	// Search correlating zone
	// Check from target window to the left until MaxFrontedgeDeviation
	ELSE
		// Calculate max number of allowed front deviation windows
		NumberOfDeviationWindows := UDINT_TO_UINT(mMaxFrontEdgeDeviation / WindowSize);
		
		// Add an additional window if rest of division was unequal 0
		IF mMaxFrontEdgeDeviation MOD WindowSize > 0 THEN
			NumberOfDeviationWindows := NumberOfDeviationWindows + 1;
		END_IF
		
		// Get max tracking position for valid zone
		MaxTrackingPosition := M_GetTrackingPosition(mAbsolutePosition - mMaxFrontEdgeDeviation);

		// Search for adjacent zone
		mWindowIndex := mNewWindowIndexFE;
				
		// Check all additional windows plus begin
		FOR mIdx := 1 TO NumberOfDeviationWindows + 1 DO
			// Correct window border overflow
			IF mWindowIndex > MaxWindowIndex THEN
				mWindowIndex := mWindowIndex - MaxWindowIndex;
			END_IF
			
			// Search next zone
			IF WindowTable[mWindowIndex].ZoneIndex > 0 THEN
				DistanceToTU_End := M_GetDistanceToTU_End(mAbsolutePosition, WindowTable[mWindowIndex].ZoneIndex);
				DistanceToTU_Start := M_GetDistanceToTU_Start(mAbsolutePosition, WindowTable[mWindowIndex].ZoneIndex);
			
				// When a found zone is valid, check if edge is in valid range
				IF WindowTable[mWindowIndex].State = E_WindowTrackingWindowState.Front_EDGE THEN
					// Check if it's not last deviation window to check
					IF mIdx < NumberOfDeviationWindows + 1 THEN
						// Return found zone
						ZoneIndex := WindowTable[mWindowIndex].ZoneIndex;
					ELSE
						// Check position in window for max deviation
						IF WindowTable[mWindowIndex].TU_FrontEdgePosition <= MaxTrackingPosition THEN			
							// Return found zone
							ZoneIndex := WindowTable[mWindowIndex].ZoneIndex;
						END_IF
					END_IF
					EXIT;
					
				// Ensure TU end has not passed resync position and TU begin has reacher in minimum MaxDeviation pos
				// Remark: >0 = It is infront of resync position 
				ELSIF DistanceToTU_End > 0 AND
					  DistanceToTU_Start <= UDINT_TO_DINT(mMaxFrontEdgeDeviation) THEN
					// Return found zone
					ZoneIndex := WindowTable[mWindowIndex].ZoneIndex;
					EXIT;
				END_IF
			END_IF
			
			mWindowIndex := mWindowIndex + 1;
		END_FOR 
	END_IF
END_IF

// Ensure zone is valid (Consists of a TU, adaption of FE possible)
IF ZoneIndex > 0 THEN
	// Only possible if zone consists of a physical TU
	IF ZoneTable[ZoneIndex].TU_Present THEN
		// Ensure that no other zone is between new front edge and old rear edge
		mWindowIndex := mNewWindowIndexFE;
		ResyncPossible := TRUE;
		
		// Calculate new zone length in windows
		IF ZoneTable[ZoneIndex].ZoneEndWindowIndex > mNewWindowIndexFE THEN
			mNewZoneWindowLength := ZoneTable[ZoneIndex].ZoneEndWindowIndex - mNewWindowIndexFE + 1;
		ELSE
			mNewZoneWindowLength := ZoneTable[ZoneIndex].ZoneEndWindowIndex + MaxWindowIndex - mNewWindowIndexFE + 1;
		END_IF
	
		// Ensure resync has space
		FOR mIdx := 1 TO mNewZoneWindowLength DO	
			// If found window is empty or already part of the zone
			IF WindowTable[mWindowIndex].ZoneIndex = 0 OR
			   WindowTable[mWindowIndex].ZoneIndex = ZoneIndex THEN
			   // Window is valid
			   ;
			
			// Otherwise another zone is found, try to shift
			ELSE
				mZoneFreeOk := M_MakeSpace(
									mStartWindowIndex 	:= mWindowIndex, 
									mWindowsToFree 		:= 1,
									mAllowZoneDelete 	:= TRUE);
									
				IF NOT mZoneFreeOk THEN
					// Error, zone could not be shifted -> abort
					ResyncPossible := FALSE;
					EXIT;
				END_IF
			END_IF
			  
			mWindowIndex := mWindowIndex + 1;

			// Correct window border overflow
			IF mWindowIndex > MaxWindowIndex THEN
				mWindowIndex := mWindowIndex - MaxWindowIndex;
			END_IF
		END_FOR  
	END_IF
END_IF

// Process when a valid zone could be found
IF ZoneIndex > 0 AND ResyncPossible THEN
	// Calculate length of existing zone in windows
	IF ZoneTable[ZoneIndex].ZoneEndWindowIndex > ZoneTable[ZoneIndex].ZoneStartWindowIndex THEN
		ZoneWindowLength := ZoneTable[ZoneIndex].ZoneEndWindowIndex - ZoneTable[ZoneIndex].ZoneStartWindowIndex + 1;
	ELSE
		ZoneWindowLength := ZoneTable[ZoneIndex].ZoneEndWindowIndex + MaxWindowIndex  - ZoneTable[ZoneIndex].ZoneStartWindowIndex + 1;
	END_IF
	
	// Get existing front edge window
	ExistingWindowIndexFE := ZoneTable[ZoneIndex].TU_StartWindowIndex;
		
	// When front edge window could be found
	IF ExistingWindowIndexFE > 0 THEN
		// Store old window, because its possible to overwrite existing position
		OldWindowFE := WindowTable[ExistingWindowIndexFE];
		M_ClearWindow(ExistingWindowIndexFE);
		
		// Copy old window to new
		WindowTable[mNewWindowIndexFE] := OldWindowFE;
		
		NewPositionFE := M_GetTrackingPosition(mAbsolutePosition);
		
		// Adapt edge position and zone length
		WindowTable[mNewWindowIndexFE].TU_FrontEdgePosition := NewPositionFE;
		ZoneTable[ZoneIndex].ZoneStartWindowIndex := mNewWindowIndexFE;
		ZoneTable[ZoneIndex].TU_StartWindowIndex := mNewWindowIndexFE;
		ZoneTable[ZoneIndex].ZoneStartPosition := NewPositionFE;
		
		IF ZoneTable[ZoneIndex].ZoneEndPosition >= ZoneTable[ZoneIndex].ZoneStartPosition THEN
			ZoneTable[ZoneIndex].ZoneLength := UDINT_TO_UINT(ZoneTable[ZoneIndex].ZoneEndPosition - ZoneTable[ZoneIndex].ZoneStartPosition);
		ELSE
			ZoneTable[ZoneIndex].ZoneLength := UDINT_TO_UINT(ZoneTable[ZoneIndex].ZoneEndPosition + TotalTrackingLength - ZoneTable[ZoneIndex].ZoneStartPosition);
		END_IF

		// Clean all windows to the right of this zone
		mWindowIndex := mNewWindowIndexFE - 1;
		
		FOR mIdx := 1 TO MaxWindowIndex DO	
			// Correct window border overflow
			IF mWindowIndex <= 0 THEN
				mWindowIndex := mWindowIndex + MaxWindowIndex;
			END_IF
			
			// When window right of the front edge is part of the same zone, clean it
			IF WindowTable[mWindowIndex].ZoneIndex = ZoneIndex THEN
				M_ClearWindow(mWindowIndex);
				mWindowIndex := mWindowIndex -1;
			// Otherwise no other windows to clean
			ELSE
				EXIT;
			END_IF
		END_FOR  
			
		// Fill gap windows to the left
		mWindowIndex := mNewWindowIndexFE;
				
		FOR mIdx := 1 TO mNewZoneWindowLength DO	
			// Correct window border overflow
			IF mWindowIndex > MaxWindowIndex THEN
				mWindowIndex := mWindowIndex - MaxWindowIndex;
			END_IF
			
			// Assign ZoneIndex to all windows
			WindowTable[mWindowIndex].ZoneIndex := ZoneIndex;
			
			// Overwrite all windows as occupied except begin and end
			IF WindowTable[mWindowIndex].State = E_WindowTrackingWindowState.FRONT_EDGE THEN
				;
			// Stop overwriting at rear edge window
            ELSIF WindowTable[mWindowIndex].State = E_WindowTrackingWindowState.REAR_EDGE THEN
				EXIT;
			ELSE
				// Assign ZoneIndex to all windows
				WindowTable[mWindowIndex].ZoneIndex := ZoneIndex;
				WindowTable[mWindowIndex].State := E_WindowTrackingWindowState.OCCUPIED;
			
				// Possible flush can be resettet, because of synchronization its valid again
				WindowTable[mWindowIndex].Flush := 0;
				WindowTable[mWindowIndex].TU_FrontEdgePosition := 0;
				WindowTable[mWindowIndex].TU_RearEdgePosition := 0;
			END_IF

			mWindowIndex := mWindowIndex + 1;
		END_FOR  
		
		M_ResyncOnlyFE := ZoneIndex;
	END_IF
END_IF
END_METHOD

/// This function synchronize only Rear edge to a specific position and calculates new TU length.
/// Remark: Zone end gets adjusted to new rear edge position. Spare windows after rear edge get removed.
/// Remark: If at absolute position no zone is found, it search to the right
/// until "mMaxFrontEdgeDeviation" to find one to synchronize.
METHOD M_ResyncOnlyRE : UINT // Returns > 0 of the synchronized Zone index, otherwise 0
VAR_INPUT
	mAbsolutePosition		: UDINT; // Absolute position [mm]
	mMaxRearEdgeDeviation 	: UDINT; (* When zone can not be found at "Absolute position",
										a search upwards is executed to a limit of MaxRearEdgeDeviation [mm]*)
END_VAR
VAR_INST
	MinTrackingPosition		: UDINT; // Min tracking distance to search for a zone
	NumberOfDeviationWindows: UINT; // Number of windows for maximal edge deviation 
	ZoneIndex				: UINT; // Zone index
	ResyncPossible			: BOOL; // Resync is possible
	ExistingWindowIndexRE	: UINT; // Existing rear edge window index
	ZoneWindowLength 		: UINT; // Length of zone to be moved
	OldWindowRE				: ST_WindowTrackingWindow; // Stored old rear edge window
	NewPositionRE			: UDINT; // New rear edge position in tracking
	DistanceToTU_End		: DINT; // Distance to found TU End
	DistanceToTU_Start		: DINT; // Distance to found TU start
END_VAR
VAR
	mZoneFreeOk				: BOOL; // Successfully
	mNewZoneWindowLength	: UINT; // Length of windows of aligned zone
	mNewWindowIndexRE		: UINT; // Actual window index
	mWindowIndex			: UINT; // Window index iterator
	mIdx					: UINT; // Loop iterator
END_VAR
M_ResyncOnlyRE := 0;
ZoneIndex := 0;
NumberOfDeviationWindows := 0;

// Validate values
IF WindowSize = 0 THEN
	RETURN;
END_IF

// Get window index at position
mNewWindowIndexRE := M_GetWindowIndex(mAbsolutePosition);

IF mNewWindowIndexRE > 0 AND mNewWindowIndexRE <= WindowTracking.MAX_NUMBER_OF_WINDOWS THEN
	// Ensure that target window is not already a front edge window 
	// This is not permitted, minimum zone is two window
	IF WindowTable[mNewWindowIndexRE].State = E_WindowTrackingWindowState.FRONT_EDGE THEN
		ZoneIndex := 0;
		
	// Search correlating zone
	// Check from target window to the right until MaxFrontedgeDeviation
	ELSE
		// Calculate max number of allowed rear edge deviation windows
		NumberOfDeviationWindows := UDINT_TO_UINT(mMaxRearEdgeDeviation / WindowSize);
		
		// Add an additional window if rest of division was unequal 0
		IF mMaxRearEdgeDeviation MOD WindowSize > 0 THEN
			NumberOfDeviationWindows := NumberOfDeviationWindows + 1;
		END_IF
		
		// Get min  tracking position for valid zone
		MinTrackingPosition := M_GetTrackingPosition(mAbsolutePosition + mMaxRearEdgeDeviation);

		// Search for a adjacent zone
		mWindowIndex := mNewWindowIndexRE;

		FOR mIdx := 1 TO NumberOfDeviationWindows + 1 DO	
			// Correct window border overflow
			IF mWindowIndex <= 0 THEN
				mWindowIndex := mWindowIndex + MaxWindowIndex;
			END_IF
			
			// Search next zone
			IF WindowTable[mWindowIndex].ZoneIndex > 0 THEN
				DistanceToTU_End := M_GetDistanceToTU_End(mAbsolutePosition, WindowTable[mWindowIndex].ZoneIndex);
				DistanceToTU_Start := M_GetDistanceToTU_Start(mAbsolutePosition, WindowTable[mWindowIndex].ZoneIndex);
			
				// When a rear edge was found check for valid range
				IF WindowTable[mWindowIndex].State = E_WindowTrackingWindowState.REAR_EDGE THEN
					// If it's not last deviation window to check
					IF mIdx < NumberOfDeviationWindows + 1 THEN
						// Return found zone
						ZoneIndex := WindowTable[mWindowIndex].ZoneIndex;
					ELSE
						// Check position in window for max deviation
						IF WindowTable[mWindowIndex].TU_RearEdgePosition >= MinTrackingPosition THEN			
							// Return found zone
							ZoneIndex := WindowTable[mWindowIndex].ZoneIndex;
						END_IF
					END_IF
					EXIT;
					
				// Ensure TU start has passed resync position and TU end has reached in minimum MaxDeviation pos
				// Remark: >0 = It is infront of resync position 
				ELSIF DistanceToTU_Start < 0 AND
                      DistanceToTU_End >= UDINT_TO_DINT(mMaxRearEdgeDeviation) THEN
				   	// Return found zone
					ZoneIndex := WindowTable[mWindowIndex].ZoneIndex;
					EXIT;
				END_IF
			END_IF
			
			mWindowIndex := mWindowIndex - 1;
		END_FOR 
	END_IF
END_IF

// Ensure zone is valid (Consists of a TU, adaption of RE possible)
IF ZoneIndex > 0 THEN
	// Only possible if zone consists of a physical TU
	IF ZoneTable[ZoneIndex].TU_Present THEN
		// Ensure that no other zone is between new rear edge and old front edge
		mWindowIndex := ZoneTable[ZoneIndex].ZoneStartWindowIndex;
		ResyncPossible := TRUE;
		
		// Calculate new zone length in windows
		IF mNewWindowIndexRE > ZoneTable[ZoneIndex].ZoneStartWindowIndex THEN
			mNewZoneWindowLength := mNewWindowIndexRE - ZoneTable[ZoneIndex].ZoneStartWindowIndex + 1;
		ELSE
			mNewZoneWindowLength := mNewWindowIndexRE  + MaxWindowIndex - ZoneTable[ZoneIndex].ZoneStartWindowIndex + 1;
		END_IF
	
		// Validate that sync is possible
		FOR mIdx := 1 TO mNewZoneWindowLength DO	
			// If found window is empty or already part of the zone
			IF WindowTable[mWindowIndex].ZoneIndex = 0 OR
			   WindowTable[mWindowIndex].ZoneIndex = ZoneIndex THEN
			   // Window is valid
			   ;
			
			// Otherwise another zone is found, try to shift
			ELSE
				mZoneFreeOk := M_MakeSpace(
									mStartWindowIndex 	:= mWindowIndex, 
									mWindowsToFree 		:= 1,
									mAllowZoneDelete 	:= TRUE);
									
				IF NOT mZoneFreeOk THEN
					// Error, zone could not be shifted -> abort
					ResyncPossible := FALSE;
					EXIT;
				END_IF
			END_IF
			  
			mWindowIndex := mWindowIndex + 1;

			// Correct window border overflow
			IF mWindowIndex > MaxWindowIndex THEN
				mWindowIndex := mWindowIndex - MaxWindowIndex;
			END_IF
		END_FOR  
	END_IF
END_IF

IF ZoneIndex > 0 AND ResyncPossible THEN
	// Calculate length of existing zone in windows
	IF ZoneTable[ZoneIndex].ZoneEndWindowIndex > ZoneTable[ZoneIndex].ZoneStartWindowIndex THEN
		ZoneWindowLength := ZoneTable[ZoneIndex].ZoneEndWindowIndex - ZoneTable[ZoneIndex].ZoneStartWindowIndex + 1;
	ELSE
		ZoneWindowLength := ZoneTable[ZoneIndex].ZoneEndWindowIndex + MaxWindowIndex  - ZoneTable[ZoneIndex].ZoneStartWindowIndex + 1;
	END_IF
	
	// Get existing rear edge window
	ExistingWindowIndexRE := ZoneTable[ZoneIndex].TU_EndWindowIndex;
	
	// When rear edge window could be found
	IF ExistingWindowIndexRE > 0 THEN
		// Store old window, because its possible to overwrite existing position
		OldWindowRE := WindowTable[ExistingWindowIndexRE];
		M_ClearWindow(ExistingWindowIndexRE);
		
		// Copy old window to new
		WindowTable[mNewWindowIndexRE] := OldWindowRE;
		
		NewPositionRE := M_GetTrackingPosition(mAbsolutePosition);
		
		// Adapt edge position and zone length
		WindowTable[mNewWindowIndexRE].TU_RearEdgePosition := NewPositionRE;
		ZoneTable[ZoneIndex].ZoneEndWindowIndex := mNewWindowIndexRE;
		ZoneTable[ZoneIndex].TU_EndWindowIndex := mNewWindowIndexRE;
		ZoneTable[ZoneIndex].ZoneEndPosition := NewPositionRE;
		
		IF ZoneTable[ZoneIndex].ZoneEndPosition >= ZoneTable[ZoneIndex].ZoneStartPosition THEN
			ZoneTable[ZoneIndex].ZoneLength := UDINT_TO_UINT(ZoneTable[ZoneIndex].ZoneEndPosition - ZoneTable[ZoneIndex].ZoneStartPosition);
		ELSE
			ZoneTable[ZoneIndex].ZoneLength := UDINT_TO_UINT(ZoneTable[ZoneIndex].ZoneEndPosition + TotalTrackingLength - ZoneTable[ZoneIndex].ZoneStartPosition);
		END_IF
		
		// Clean all windows to the left of this zone
		mWindowIndex := mNewWindowIndexRE + 1;
		
		FOR mIdx := 1 TO MaxWindowIndex DO	
			// Correct window border overflow
			IF mWindowIndex > MaxWindowIndex THEN
				mWindowIndex := mWindowIndex - MaxWindowIndex;
			END_IF
			
			// When window left of the rear edge is part of the same zone, clean it
			IF WindowTable[mWindowIndex].ZoneIndex = ZoneIndex THEN
				M_ClearWindow(mWindowIndex);
				mWindowIndex := mWindowIndex + 1;
			// Otherwise no other windows to clean
			ELSE
				EXIT;
			END_IF
		END_FOR  
			
		// Fill gap windows to the right
		mWindowIndex := mNewWindowIndexRE;
				
		FOR mIdx := 1 TO mNewZoneWindowLength DO	
			// Correct window border overflow
			IF mWindowIndex <= 0 THEN
				mWindowIndex := mWindowIndex + MaxWindowIndex;
			END_IF
			
			// Assign ZoneIndex to all windows
			WindowTable[mWindowIndex].ZoneIndex := ZoneIndex;
			
			// Overwrite all windows as occupied except begin and end
			IF WindowTable[mWindowIndex].State = E_WindowTrackingWindowState.REAR_EDGE THEN
				;
				
			// Stop overwriting at front edge window
            ELSIF WindowTable[mWindowIndex].State = E_WindowTrackingWindowState.FRONT_EDGE THEN
				EXIT;
				
			ELSE
				// Assign ZoneIndex to all windows
				WindowTable[mWindowIndex].ZoneIndex := ZoneIndex;
				WindowTable[mWindowIndex].State := E_WindowTrackingWindowState.OCCUPIED;
			
				// Possible flush can be reset, because of synchronization its valid again
				WindowTable[mWindowIndex].Flush := 0;
				WindowTable[mWindowIndex].TU_FrontEdgePosition := 0;
				WindowTable[mWindowIndex].TU_RearEdgePosition := 0;
			END_IF

			mWindowIndex := mWindowIndex - 1;
		END_FOR  
		
		M_ResyncOnlyRE := ZoneIndex;
	END_IF
END_IF
END_METHOD

/// This function synchronize whole TU aligned by Front edge to a specific position.
/// Rear edge is adjusted automatically to keep the length of TU.
/// Remark: If at absolute position no zone is found, it search to the left
/// until "mMaxFrontEdgeDeviation" to find one to synchronize.
METHOD M_ResyncTU_FE : UINT // Returns > 0 of the synchronized Zone index, otherwise 0
VAR_INPUT
	mAbsolutePosition		: UDINT; // Absolute position [mm]
	mMaxFrontEdgeDeviation 	: UDINT; (* When zone can not be found at "Absolute position",
										a search upwards is executed to a limit of MaxFrontEdgeDeviation [mm]*)
END_VAR
VAR_INST
	MaxTrackingPosition		: UDINT; // Max tracking distance to search for a zone
	NumberOfDeviationWindows: UINT; // Number of windows for maximal edge deviation 
	ZoneIndex				: UINT; // Zone index
END_VAR
VAR
	mZoneMoved 				: BOOL; // Zone moved successfully
	mSyncWindowIndex		: UINT; // Actual window index
	mWindowIndex			: UINT; // Window index iterator
	mIdx					: UINT; // Loop iterator
	DistanceToTU_End		: DINT; // Distance to found TU End
	DistanceToTU_Start		: DINT; // Distance to found TU start
END_VAR
M_ResyncTU_FE := 0;
ZoneIndex := 0;
NumberOfDeviationWindows := 0;

// Validate values
IF WindowSize = 0 THEN
	RETURN;
END_IF

// Get window index at position
mSyncWindowIndex := M_GetWindowIndex(mAbsolutePosition);

// Search correlating zone
// Check from target window to the left until MaxFrontedgeDeviation
IF mSyncWindowIndex > 0 AND mSyncWindowIndex <= WindowTracking.MAX_NUMBER_OF_WINDOWS THEN
	// Calculate max number of allowed front deviation windows
	NumberOfDeviationWindows := UDINT_TO_UINT(mMaxFrontEdgeDeviation / WindowSize);
	
	// Add an additional window if rest of division was unequal 0
	IF mMaxFrontEdgeDeviation MOD WindowSize > 0 THEN
		NumberOfDeviationWindows := NumberOfDeviationWindows + 1;
	END_IF
	
	// Get max tracking position for valid zone
	MaxTrackingPosition := M_GetTrackingPosition(mAbsolutePosition - mMaxFrontEdgeDeviation);

	// Search for adjacent zone
	mWindowIndex := mSyncWindowIndex;
			
	FOR mIdx := 1 TO NumberOfDeviationWindows + 1 DO	
		// Correct window border overflow
		IF mWindowIndex > MaxWindowIndex THEN
			mWindowIndex := mWindowIndex - MaxWindowIndex;
		END_IF
		
		// Search next zone
		IF WindowTable[mWindowIndex].ZoneIndex > 0 THEN
			DistanceToTU_End := M_GetDistanceToTU_End(mAbsolutePosition, WindowTable[mWindowIndex].ZoneIndex);
			DistanceToTU_Start := M_GetDistanceToTU_Start(mAbsolutePosition, WindowTable[mWindowIndex].ZoneIndex);
			
			// When a found zone is valid, check if edge is in valid range
			IF WindowTable[mWindowIndex].State = E_WindowTrackingWindowState.Front_EDGE THEN
				// Check if it's not last deviation window to check
				// Then it is anyway in the valid range
				IF mIdx < NumberOfDeviationWindows + 1 THEN
					// Return found zone
					ZoneIndex := WindowTable[mWindowIndex].ZoneIndex;
					
				// if it is the last window,
				// ensure the position inside the window is in the allowed border
				ELSE
					// Check position in window for max deviation
					IF WindowTable[mWindowIndex].TU_FrontEdgePosition <= MaxTrackingPosition THEN			
						// Return found zone
						ZoneIndex := WindowTable[mWindowIndex].ZoneIndex;
					END_IF
				END_IF
				EXIT;
				
			// Ensure TU end has not passed resync position and TU begin has reacher in minimum MaxDeviation pos
			// Remark: >0 = It is infront of resync position 
			ELSIF DistanceToTU_End > 0 AND
                  DistanceToTU_Start <= UDINT_TO_DINT(mMaxFrontEdgeDeviation) THEN
				// Return found zone
				ZoneIndex := WindowTable[mWindowIndex].ZoneIndex;
				EXIT;
			END_IF
		END_IF
		
		mWindowIndex := mWindowIndex + 1;
	END_FOR 
END_IF

// Process when a zone could be found
IF ZoneIndex > 0 THEN
	mZoneMoved := M_MoveZoneFE(
					mZoneIndex 				:= ZoneIndex,
					mAbsoluteTargetPosition := mAbsolutePosition,
					mDeleteTargetZones 		:= FALSE);
					
	IF mZoneMoved THEN
		M_ResyncTU_FE := ZoneIndex;
	ELSE
		M_ResyncTU_FE := 0;
	END_IF
END_IF
END_METHOD

/// This function synchronize whole TU aligned by Rear edge to a specific position.
/// Front edge is adjusted automatically to keep the length of TU.
/// Remark: If at absolute position no zone is found, it search to the right
/// until "mMaxFrontEdgeDeviation" to find one to synchronize.
METHOD M_ResyncTU_RE : UINT // Returns > 0 of the synchronized Zone index, otherwise 0
VAR_INPUT
	mAbsolutePosition		: UDINT; // Absolute position [mm]
	mMaxRearEdgeDeviation 	: UDINT; (* When zone can not be found at "Absolute position",
										a search upwards is executed to a limit of MaxRearEdgeDeviation [mm]*)
END_VAR
VAR_INST
	MinTrackingPosition		: UDINT; // Min tracking distance to search for a zone
	NumberOfDeviationWindows: UINT; // Number of windows for maximal edge deviation 
	ZoneIndex				: UINT; // Zone index
	DistanceToTU_End		: DINT; // Distance to found TU End
	DistanceToTU_Start		: DINT; // Distance to found TU start
END_VAR
VAR
	mZoneMoved 				: BOOL; // Zone moved successfully
	mSyncWindowIndex		: UINT; // Actual window index
	mWindowIndex			: UINT; // Window index iterator
	mIdx					: UINT; // Loop iterator
END_VAR
M_ResyncTU_RE := 0;
ZoneIndex := 0;
NumberOfDeviationWindows := 0;

// Validate values
IF WindowSize = 0 THEN
	RETURN;
END_IF

// Get window index at position
mSyncWindowIndex := M_GetWindowIndex(mAbsolutePosition);

IF mSyncWindowIndex > 0 AND mSyncWindowIndex <= WindowTracking.MAX_NUMBER_OF_WINDOWS THEN
	// Calculate max number of allowed rear edge deviation windows
	NumberOfDeviationWindows := UDINT_TO_UINT(mMaxRearEdgeDeviation / WindowSize);
	
	// Add an additional window if rest of division was unequal 0
	IF mMaxRearEdgeDeviation MOD WindowSize > 0 THEN
		NumberOfDeviationWindows := NumberOfDeviationWindows + 1;
	END_IF
	
	// Get min tracking position for valid zone
	MinTrackingPosition := M_GetTrackingPosition(mAbsolutePosition - mMaxRearEdgeDeviation);

	// Search for a adjacent zone to the right
	mWindowIndex := mSyncWindowIndex;
			
	FOR mIdx := 1 TO NumberOfDeviationWindows + 1 DO	
		// Correct window border overflow
		IF mWindowIndex <= 0 THEN
			mWindowIndex := mWindowIndex + MaxWindowIndex;
		END_IF
		
		// Search next zone
		IF WindowTable[mWindowIndex].ZoneIndex > 0 THEN
			DistanceToTU_End := M_GetDistanceToTU_End(mAbsolutePosition, WindowTable[mWindowIndex].ZoneIndex);
			DistanceToTU_Start := M_GetDistanceToTU_Start(mAbsolutePosition, WindowTable[mWindowIndex].ZoneIndex);
			
			// When a found zone is valid, check if edge is in valid range
			IF WindowTable[mWindowIndex].State = E_WindowTrackingWindowState.REAR_EDGE THEN
				// If it's not last deviation window to check
				IF mIdx < NumberOfDeviationWindows THEN
					// Return found zone
					ZoneIndex := WindowTable[mWindowIndex].ZoneIndex;
				ELSE
					// Check position in window for max deviation
					IF WindowTable[mWindowIndex].TU_RearEdgePosition >= MinTrackingPosition THEN
						// Return found zone
						ZoneIndex := WindowTable[mWindowIndex].ZoneIndex;
					END_IF
				END_IF
				EXIT;
				
			// Ensure TU start has passed resync position and TU end has reached in minimum MaxDeviation pos
			// Remark: >0 = It is infront of resync position 
			ELSIF DistanceToTU_Start < 0 AND
                  DistanceToTU_End >= UDINT_TO_DINT(mMaxRearEdgeDeviation) THEN
				 // Return found zone
				ZoneIndex := WindowTable[mWindowIndex].ZoneIndex;
				EXIT;
			END_IF
		END_IF
		
		mWindowIndex := mWindowIndex - 1;
	END_FOR 
END_IF

// Process when a zone could be found
IF ZoneIndex > 0 THEN
	mZoneMoved := M_MoveZoneRE(
					mZoneIndex 				:= ZoneIndex,
					mAbsoluteTargetPosition := mAbsolutePosition,
					mDeleteTargetZones 		:= FALSE);
					
	IF mZoneMoved THEN
		M_ResyncTU_RE := ZoneIndex;
	ELSE
		M_ResyncTU_RE := 0;
	END_IF
END_IF
END_METHOD

/// Shift zone at StartWindowIndex by WindowsToShift (If WindowsToShift includes more zones, they are shifted as well)
/// Remark: Only Zones without a TU Present and permition to shift, can be shifted. 
/// Remark: When a zone is found to shift, the whole zone is shifted
/// Remark: Zones which can not be reallocated (e.g. not enough space on tracking) get deleted. Owner of the Zone
/// will be notfied about that process.
METHOD PROTECTED M_ShiftZone : BOOL // Returns true if successfull shifted, otherwise false (e.g. not allowed to shift, wrong input)
VAR_INPUT
	mStartWindowIndex		: UINT; // Start window index
	mWindowsToShift			: UINT; // Windows to shift
	mExcludeTUs				: BOOL; // Exclude physical occupied zones
	mAllowOverrun			: BOOL; // Allow to throw out zones which cannot be place on the tracking anymore because of reallocations
END_VAR
VAR_INST
	ShiftingAllowed			: BOOL; // Target position is to be shifted
	RetrieveOk 				: BOOL; // Retrieve reallocation order successfully
	MoveOk 					: BOOL; // Move of zone executed successfully
	RelocEntry 				: ST_WindowTrackingReloc; // Reallocation order
	fbRelocator 			: FB_WindowRelocator; // Windows relocator
	ZoneOverrun				: BOOL;
	ZoneOverrunWindowIndex	: UINT;
END_VAR
VAR
	mIdx 					: DINT; // Loop iterator
	mNumberOfOverrunWindows : UINT;
	mEndOverrunWindowIndex	: UINT;
	mWindowIndex 			: UDINT; // Window index to loop trough tracking distance
END_VAR
M_ShiftZone := FALSE;

// Validate inputs
IF mStartWindowIndex = 0 OR
   mStartWindowIndex > WindowTracking.MAX_NUMBER_OF_WINDOWS OR
   mWindowsToShift = 0 OR
   mWindowsToShift > WindowTracking.MAX_NUMBER_OF_WINDOWS OR
   WindowSize = 0 THEN
	RETURN;
END_IF

// Inform listener
IF iEventListener <> 0 THEN
	iEventListener.M_TrackingShiftingInitiatedEvent(
		mAbsolutePosition 	:= M_GetAbsolutePosition(mStartWindowIndex - 1 * WindowSize),
		mDistance 			:= mWindowsToShift * WindowSize,
		mWindowIndex 		:= mStartWindowIndex,
		mWindowsToShift 	:= mWindowsToShift);
END_IF

fbRelocator.M_Reset();

ShiftingAllowed := M_IsShiftable(
						mStartWindowIndex,
						mWindowsToShift,
						mExcludeTUs,
						mAllowOverrun,
						mZoneOverrun => ZoneOverrun,
						mZoneOverrunWindowIndex => ZoneOverrunWindowIndex,
						mfbRelocator := fbRelocator);

IF ShiftingAllowed THEN
	// Clear overrun distance if allowed
	IF ZoneOverrun THEN
		IF mStartWindowIndex = 1 THEN
			mEndOverrunWindowIndex := MaxWindowIndex;
		ELSE	
			mEndOverrunWindowIndex := mStartWindowIndex - 1;
		END_IF
	
		IF mEndOverrunWindowIndex >= ZoneOverrunWindowIndex THEN
			mNumberOfOverrunWindows := mEndOverrunWindowIndex - ZoneOverrunWindowIndex;
		ELSE
			mNumberOfOverrunWindows := mEndOverrunWindowIndex + MaxWindowIndex - ZoneOverrunWindowIndex;
		END_IF
		
		mWindowIndex := ZoneOverrunWindowIndex;
		
		// Clear all zones which can not be relocated
		FOR mIdx := 1 TO mNumberOfOverrunWindows DO
			IF WindowTable[mWindowIndex].ZoneIndex > 0 THEN
				M_DeleteZone(WindowTable[mWindowIndex].ZoneIndex);
			END_IF
			
			mWindowIndex := mWindowIndex + 1;
			
			IF mWindowIndex > MaxWindowIndex THEN
				mWindowIndex := mWindowIndex - MaxWindowIndex;
			END_IF
		END_FOR
	END_IF

	// Do reallocation
	// Execute all scheduled reallocations
	FOR mIdx := 1 TO MAX_NUMBER_OF_ZONES DO
		
		RetrieveOk := fbRelocator.M_RetrieveLastEntry(
						mpData 		:= ADR(RelocEntry),
						mDataSize 	:= SIZEOF(RelocEntry));
						
		// Move all zones according all stored reallocation orders starting with the last added
		IF RetrieveOk THEN
			MoveOk := M_MoveZone(
						mZoneIndex 				:= RelocEntry.ZoneIndex,
						mTargetStartWindow 		:= RelocEntry.TargetWindow,
						mEnableDeleteOfZones 	:= TRUE);
						
			IF NOT MoveOk THEN
				// Error
				fbDebugMsg.M_SendErrorMsg('M_ShiftZone - Move was not possible.');	
			END_IF
		ELSE
			// No entries available anymore
			EXIT;
		END_IF
	END_FOR
	
	// Shifting executed
	M_ShiftZone := TRUE;
ELSE
	M_ShiftZone := FALSE;
END_IF

// Inform listener
IF iEventListener <> 0 THEN
	iEventListener.M_TrackingShiftingCompletedEvent(
		mAbsolutePosition 	:= M_GetAbsolutePosition(mStartWindowIndex - 1 * WindowSize),
		mDistance 			:= mWindowsToShift * WindowSize,
		mWindowIndex 		:= mStartWindowIndex,
		mWindowsToShift 	:= mWindowsToShift);
END_IF
END_METHOD

/// Shortens a zone by given value in up- or downstream direction
METHOD M_ShortenZone : BOOL// Returns TRUE if successful,
VAR_INPUT
	mZoneIndex 				: UINT; // Zone index to enlarge
	mReductionLength		: UINT; // Reduce existing zone by this length [mm]
	mShiftFrontEdge			: BOOL; // Shift front edge for reduction
END_VAR
VAR
	mIdx					: UINT; // Loop iterator
	mWindowIndex			: UINT; // Start window index
	mReductionWindowLength	: UINT; // Zone length in windows
	mReductionAllowed 		: BOOL; // Reduction valid
	mZoneEndWindowIndex		: UINT; // Zone end window index
	mZoneStartWindowIndex	: UINT; // Zone start window index
	mZoneEndPositionNew		: UDINT; // Zone end position after reduction
	mZoneStartPositionNew	: UDINT; // Zone start position after enlargement
END_VAR
VAR_INST
	OldZoneData				: ST_WindowTrackingZone; // Old tracking zone data
END_VAR
M_ShortenZone := FALSE;

// Validate inputs
IF mZoneIndex <= 0 OR
   mZoneIndex > MAX_NUMBER_OF_ZONES OR
   WindowSize = 0 THEN
   RETURN;
END_IF

IF ZoneTable[mZoneIndex].TU_Present THEN
	IF NOT mShiftFrontEdge THEN
		// Calculate new zone end position
		IF mReductionLength > ZoneTable[mZoneIndex].ZoneEndPosition THEN
			mZoneEndPositionNew := ZoneTable[mZoneIndex].ZoneEndPosition - mReductionLength + TotalTrackingLength;
			mReductionWindowLength := M_GetWindowIndex(M_GetAbsolutePosition(ZoneTable[mZoneIndex].ZoneEndPosition)) - M_GetWindowIndex(M_GetAbsolutePosition(mZoneEndPositionNew)) + MaxWindowIndex + 1;
		ELSE
			mZoneEndPositionNew := ZoneTable[mZoneIndex].ZoneEndPosition - mReductionLength;
			mReductionWindowLength := M_GetWindowIndex(M_GetAbsolutePosition(ZoneTable[mZoneIndex].ZoneEndPosition)) - M_GetWindowIndex(M_GetAbsolutePosition(mZoneEndPositionNew)) + 1;
		END_IF
		
		mWindowIndex := ZoneTable[mZoneIndex].ZoneEndWindowIndex;
		mReductionAllowed := TRUE;
		
		// Ensure reduction is possible
		FOR mIdx := 1 TO mReductionWindowLength DO
			// Is intended window index not occupied by TU
			IF WindowTable[mWindowIndex].State <> E_WindowTrackingWindowState.RESERVED THEN
				mReductionAllowed := FALSE;
				// Error
				fbDebugMsg.M_SendErrorMsg('M_ShortenZone - Reduction not possible, TU already in range of reduction.');	
				RETURN;
			END_IF
			
			mWindowIndex := mWindowIndex - 1;
			
			// Correct border overflow
			IF mWindowIndex = 0 THEN
				mWindowIndex := MaxWindowIndex;
			END_IF
		END_FOR
	ELSE
		// Calculate new zone start position
		IF ZoneTable[mZoneIndex].ZoneStartPosition + mReductionLength > TotalTrackingLength THEN
			mZoneStartPositionNew := ZoneTable[mZoneIndex].ZoneStartPosition + mReductionLength - TotalTrackingLength;
			mReductionWindowLength := M_GetWindowIndex(M_GetAbsolutePosition(mZoneStartPositionNew)) - M_GetWindowIndex(M_GetAbsolutePosition(ZoneTable[mZoneIndex].ZoneStartPosition)) + MaxWindowIndex + 1;
		ELSE
			mZoneStartPositionNew := ZoneTable[mZoneIndex].ZoneStartPosition + mReductionLength;
			mReductionWindowLength := M_GetWindowIndex(M_GetAbsolutePosition(mZoneStartPositionNew)) - M_GetWindowIndex(M_GetAbsolutePosition(ZoneTable[mZoneIndex].ZoneStartPosition)) + 1;
		END_IF
		
		mWindowIndex := ZoneTable[mZoneIndex].ZoneStartWindowIndex;
		mReductionAllowed := TRUE;
		
		// Ensure reduction is possible
		FOR mIdx := 1 TO mReductionWindowLength DO
			// Is intended window index not occupied by TU
			IF WindowTable[mWindowIndex].State <> E_WindowTrackingWindowState.RESERVED THEN
				mReductionAllowed := FALSE;
				// Error
				fbDebugMsg.M_SendErrorMsg('M_ShortenZone - Reduction not possible, TU already in range of reduction.');	
				RETURN;
			END_IF
			
			mWindowIndex := mWindowIndex + 1;
			
			// Correct border overflow
			IF mWindowIndex > MaxWindowIndex THEN
				mWindowIndex := mWindowIndex - MaxWindowIndex;
			END_IF
		END_FOR
	END_IF
END_IF

// When reduction is possible to be executed
IF mReductionAllowed THEN
	OldZoneData := ZoneTable[mZoneIndex];
	
	IF NOT mShiftFrontEdge THEN
		mWindowIndex := ZoneTable[mZoneIndex].ZoneEndWindowIndex;
	
		// Loop through all windows and assign new zone
		// Init
		mZoneEndWindowIndex := mWindowIndex;
		
		FOR mIdx := 1 TO mReductionWindowLength DO
			// Clear window
			MEMSET(ADR(WindowTable[mWindowIndex]), 0, SIZEOF(WindowTable[mWindowIndex]));
			
			mWindowIndex := mWindowIndex - 1;
			
			// Correct border overflow
			IF mWindowIndex = 0 THEN
				mWindowIndex := MaxWindowIndex;
			END_IF
				
			mZoneEndWindowIndex := mWindowIndex;
		END_FOR	
		
		// Update zone table
		ZoneTable[mZoneIndex].ZoneEndWindowIndex := mZoneEndWindowIndex;
		ZoneTable[mZoneIndex].ZoneEndPosition := mZoneEndPositionNew;
		ZoneTable[mZoneIndex].ZoneLength := ZoneTable[mZoneIndex].ZoneLength - mReductionLength;
		
		// Inform listener
		IF iEventListener <> 0 THEN
			iEventListener.M_TrackingZoneShortenedEvent(
				mTrackingZoneIndex 		:= mZoneIndex,
                mOldTrackingZoneData 	:= OldZoneData,
                mNewTrackingZoneDAta 	:= ZoneTable[mZoneIndex]);
		END_IF

		M_ShortenZone := TRUE;
	ELSE
		mWindowIndex := ZoneTable[mZoneIndex].ZoneStartWindowIndex;
	
		// Loop through all windows and assign new zone
		// Init
		mZoneStartWindowIndex := mWindowIndex;
		
		FOR mIdx := 1 TO mReductionWindowLength DO
			// Clear window
			MEMSET(ADR(WindowTable[mWindowIndex]), 0, SIZEOF(WindowTable[mWindowIndex]));
			
			mWindowIndex := mWindowIndex + 1;
			
			// Correct border overflow
			IF mWindowIndex > MaxWindowIndex THEN
				mWindowIndex := mWindowIndex - MaxWindowIndex;
			END_IF
				
			mZoneStartWindowIndex := mWindowIndex;
		END_FOR	
		
		// Update zone table
		ZoneTable[mZoneIndex].ZoneStartWindowIndex := mZoneStartWindowIndex;
		ZoneTable[mZoneIndex].ZoneStartPosition := mZoneStartPositionNew;
		ZoneTable[mZoneIndex].ZoneLength := ZoneTable[mZoneIndex].ZoneLength - mReductionLength;
		
		// Inform listener
		IF iEventListener <> 0 THEN
			iEventListener.M_TrackingZoneShortenedEvent(
				mTrackingZoneIndex 		:= mZoneIndex,
                mOldTrackingZoneData 	:= OldZoneData,
                mNewTrackingZoneDAta 	:= ZoneTable[mZoneIndex]);
		END_IF
		
		M_ShortenZone := TRUE;
	END_IF
END_IF
END_METHOD

/// Shortes a zone from window to its boder where no TU is in between
METHOD PROTECTED M_ShortenZoneAtWindow : BOOL // Returns true if successful, otherwise false
VAR_INPUT
	mZoneIndex			: UINT;
	mWindowIndex		: UINT; // Start window index
END_VAR
VAR_INST
	ShortenAfterTU 		: BOOL; // Shorten on side between zone end and tu end
	ShortenInFrontOfTU 	: BOOL; // Shorten on side between tu start and zone start
	ShortenLengthMM		: UINT; // Length to shorten
END_VAR
M_ShortenZoneAtWindow := FALSE;
ShortenAfterTU:= FALSE;
ShortenInFrontOfTU := FALSE;
ShortenLengthMM := 0;

// Validate inputs
IF mWindowIndex = 0 OR
   mWindowIndex > WindowTracking.MAX_NUMBER_OF_WINDOWS OR 
   mZoneIndex = 0 THEN
	RETURN;
END_IF
 
IF WindowTable[mWindowIndex].ZoneIndex <> mZoneIndex THEN
	RETURN;
END_IF

IF ZoneTable[mZoneIndex].TU_Present THEN
	// Find related border (No TU between window index and border)
	//        |
	//        v     TU
	//            ||||||
	//   |--------||||||----|
	//   

	// Check for no overflow between zone end and tu rear edge
	IF ZoneTable[mZoneIndex].ZoneEndWindowIndex >= ZoneTable[mZoneIndex].TU_EndWindowIndex THEN
		// Check if window index is between
		IF mWindowIndex >= ZoneTable[mZoneIndex].TU_EndWindowIndex AND
		   mWindowIndex <= ZoneTable[mZoneIndex].ZoneEndWindowIndex THEN
		   // Window for shorten found
		   ShortenAfterTU := TRUE;
		   ShortenLengthMM := UDINT_TO_UINT(ZoneTable[mZoneIndex].ZoneEndPosition - ((mWindowIndex-1) * WindowSize));
		END_IF
	ELSE
		// Check if window index is between
		IF mWindowIndex >= ZoneTable[mZoneIndex].TU_EndWindowIndex THEN
		   	// Window for shorten found
		  	ShortenAfterTU := TRUE;
		   	ShortenLengthMM := UDINT_TO_UINT(ZoneTable[mZoneIndex].ZoneEndPosition + TotalTrackingLength - ((mWindowIndex-1) * WindowSize));
			
		ELSIF mWindowIndex <= ZoneTable[mZoneIndex].ZoneEndWindowIndex THEN
			// Window for shorten found
		   	ShortenAfterTU := TRUE;
		   	ShortenLengthMM := UDINT_TO_UINT(ZoneTable[mZoneIndex].ZoneEndPosition - ((mWindowIndex-1) * WindowSize));	
		END_IF
	END_IF
	
	// Check for no overflow between zone end and tu rear edge
	IF ZoneTable[mZoneIndex].TU_StartWindowIndex >= ZoneTable[mZoneIndex].ZoneStartWindowIndex THEN
		// Check if window index is between
		IF mWindowIndex >= ZoneTable[mZoneIndex].ZoneStartWindowIndex AND
		   mWindowIndex <= ZoneTable[mZoneIndex].TU_StartWindowIndex THEN
		   // Window for shorten found
		   ShortenInFrontOfTU := TRUE;
		   ShortenLengthMM := UDINT_TO_UINT((mWindowIndex * WindowSize) - ZoneTable[mZoneIndex].ZoneStartPosition);
		END_IF
	ELSE
		// Check if window index is between
		IF mWindowIndex >= ZoneTable[mZoneIndex].ZoneStartWindowIndex THEN
		   	// Window for shorten found
		   	ShortenInFrontOfTU := TRUE;
		   	ShortenLengthMM := UDINT_TO_UINT((mWindowIndex * WindowSize) - ZoneTable[mZoneIndex].ZoneStartPosition);
		   
		ELSIF mWindowIndex <= ZoneTable[mZoneIndex].TU_StartWindowIndex THEN
			// Window for shorten found
		   	ShortenInFrontOfTU := TRUE;
		   	ShortenLengthMM := UDINT_TO_UINT((mWindowIndex * WindowSize) + TotalTrackingLength - ZoneTable[mZoneIndex].ZoneStartPosition);
		END_IF
	END_IF

	// When window was found inside a valid area of the zone
	IF ShortenInFrontOfTU OR ShortenAfterTU THEN
		IF ShortenInFrontOfTU THEN
			M_ShortenZoneAtWindow := M_ShortenZone(mZoneIndex, ShortenLengthMM, TRUE);
	  	ELSE
			M_ShortenZoneAtWindow := M_ShortenZone(mZoneIndex, ShortenLengthMM, FALSE);
		END_IF
	END_IF
END_IF
END_METHOD

/// All Zones get deleted if they completly (Rear edge) left TrackingLength
/// Default: Enabled
PROPERTY P_DeleteZoneTrackingEnd : BOOL // Returns true if enabled, otherwise false
GET
P_DeleteZoneTrackingEnd := DeleteZoneTrackingEnd;
END_GET
SET
DeleteZoneTrackingEnd := P_DeleteZoneTrackingEnd;
END_SET
END_PROPERTY

/// Additional tracking length. Can be used to allow more additional space for reservations.
PROPERTY P_TrackingAddition : UDINT // Additional tracking distance
GET
P_TrackingAddition := TrackingAddition;
END_GET
SET
TrackingAddition := P_TrackingAddition;
END_SET
END_PROPERTY

/// Access to Ongoing trasfer list  for read operations
/// Remark: User has to ensure that writing does not influence the process in a bad way.
{attribute 'suppress_wrn_C0410'}
PROPERTY P_TransferList : REFERENCE TO ARRAY[1..TRANSFER_TABLE_SIZE] OF ST_WindowTrackingTransfer
GET
P_TransferList REF= OngoingTransferList;
END_GET
END_PROPERTY

/// Returns currently available amount of TUs
PROPERTY P_TU_Count : INT
GET
P_TU_Count := TU_Count;
END_GET
END_PROPERTY

/// Access to Window table  for read operations
/// Remark: User has to ensure that writing does not influence the process in a bad way.
{attribute 'suppress_wrn_C0410'}
PROPERTY P_WindowTable : REFERENCE TO ARRAY[1..WindowTracking.MAX_NUMBER_OF_WINDOWS] OF ST_WindowTrackingWindow;
GET
P_WindowTable REF= WindowTable;
END_GET
END_PROPERTY

/// Returns currently available amount of Zones
PROPERTY P_ZoneCount : INT
GET
P_ZoneCount := ZoneCount;
END_GET
END_PROPERTY

/// Access to Zone table  for read operations
/// Remark: User has to ensure that writing does not influence the process in a bad way.
{attribute 'suppress_wrn_C0410'}
PROPERTY P_ZoneTable : REFERENCE TO ARRAY[1..WindowTracking.MAX_NUMBER_OF_ZONES] OF ST_WindowTrackingZone;
GET
P_ZoneTable REF= ZoneTable;
END_GET
END_PROPERTY

END_FUNCTION_BLOCK

// ---- 20_Product/30_Toolbox/99_Misc/13_Helper/FB_EncoderMonitor.TcPOU
/// This function block checks that the encoder steps are valid.
/// Could be used to detect if encoder does not follow a drive. (e.g. detached encoder)
FUNCTION_BLOCK FB_EncoderMonitor
(************************************************************************************** 
* 	Application 		: BoxControl Framework 
* 	Revision 			: $Revision: 408723 $ 
* 	Revision date 		: $Date: 2018-06-27 13:49:08 +0200 (Wed, 27 Jun 2018) $ 
* 	Last changed by 	: $Author: b7bolm $ 
* 	URL 				: $URL: http://almscdc.swisslog.com/repo/SWPD/Development/BoxControlFramework/21_Projects/BCF_2.0/trunk/BCF/BCF/JumpStart/20_Product/10_App/12_E_Functions/10_Lib/10_Conv/FB_FunctionList.TcPOU $ 
* ------------------------------------------------------------------------------------ 
* 	© Swisslog AG 
* 	Swisslog is not liable for any usage of this source code that is not agreed 
* 	on between Swisslog and the other party. The mandatory legal liability remains 
* 	unaffected. 
* ------------------------------------------------------------------------------------ 
* 	Revision History: 
* 
* 	VERSION 		DATE 			INITIALS 			DESCRIPTION 
* 	0.1 			22.08.2018 		ale					First implementation
*	0.2				21.09.2018		mbo					Moved and adjusted for standard
* 
**************************************************************************************)
VAR_INPUT
	DriveRunning			: BOOL; // Drive is running (Rising edge resets error)
	EncoderValue			: UDINT; // Encoder values [increment]
	MinValueChange			: UDINT; // Minimum value change expected if drive is running
	DelayMonitoringTime		: TIME; // Time after the value change is expected
	MaxEncoderValue			: UDINT; // Max value of input "EncoderValue" Remark: Used to detect overflow, needs to be less than DINT size [increment]
	FailureThreshold		: INT; // Amount of detected failure values before an error is raised
END_VAR
VAR_OUTPUT
	Active					: BOOL; // Monitoring active
	EncoderError			: BOOL; // Encoder issue
END_VAR
VAR
	fbDelayMonitoring		: TON; // Delay encoder monitoring (e.g. ramp up)
	fbRunTrig				: R_Trig; // Rising edge detection
	DeltaEncoderValue		: DINT; // Delta encoder value 
	LastEncoderValue		: UDINT; // Last encoder value [increment]
	LastMinValueChange		: UDINT; // Last minimum value change expected
	FailureCounter			: INT; // Detected encoder error in a serie
END_VAR

fbRunTrig(CLK := DriveRunning );

// Reset error
IF fbRunTrig.Q THEN
	EncoderError := FALSE;
	FailureCounter := 0;
END_IF

// Restart delay monitoring
IF fbRunTrig.Q OR MinValueChange <> LastMinValueChange THEN
	fbDelayMonitoring(IN := FALSE);	
END_IF

fbDelayMonitoring(IN := NOT EncoderError AND DriveRunning, PT := DelayMonitoringTime);

// Create internal encoder to make movement independent from encoder overflow
DeltaEncoderValue := UDINT_TO_DINT(EncoderValue) - UDINT_TO_DINT(LastEncoderValue);

IF ABS(DeltaEncoderValue) > UDINT_TO_DINT(MaxEncoderValue/2) THEN
	// Correction with + 1 is to include the 0 in MaxEncoderValue
	IF DeltaEncoderValue < 0 THEN
		DeltaEncoderValue := DeltaEncoderValue + UDINT_TO_DINT(MaxEncoderValue) + 1;
	ELSE
		DeltaEncoderValue := UDINT_TO_DINT(EncoderValue) - (UDINT_TO_DINT(LastEncoderValue) + UDINT_TO_DINT(MaxEncoderValue)) - 1;
	END_IF
END_IF

LastEncoderValue := EncoderValue;

IF fbDelayMonitoring.Q THEN
	//Check if minimum delta step is greather than MinValueChange
	IF ABS(DeltaEncoderValue) >= UDINT_TO_DINT(ABS(MinValueChange)) THEN
		// Encoder works fine
		FailureCounter := 0;
		
	// Encoder issue found
	ELSE
		IF FailureCounter >= FailureThreshold THEN 
			EncoderError := TRUE;
		ELSE
			FailureCounter := FailureCounter + 1;
		END_IF
	END_IF
END_IF

LastMinValueChange := MinValueChange;
Active := fbDelayMonitoring.Q;

END_FUNCTION_BLOCK

// ---- 20_Product/30_Toolbox/99_Misc/13_Helper/FB_FindTrackingZones.TcPOU
// Function block searches all available tracking zones in range (Max 5 zones).
// This function block can be used to get how accurate a tu is positioned in a zone
FUNCTION_BLOCK FB_FindTrackingZones
(************************************************************************************** 
* 	Application 		: BoxControl Framework 
* 	Revision 			: $Revision: 408723 $ 
* 	Revision date 		: $Date: 2018-06-27 13:49:08 +0200 (Wed, 27 Jun 2018) $ 
* 	Last changed by 	: $Author: b7bolm $ 
* 	URL 				: $URL: http://almscdc.swisslog.com/repo/SWPD/Development/BoxControlFramework/21_Projects/BCF_2.0/trunk/BCF/BCF/JumpStart/20_Product/10_App/12_E_Functions/10_Lib/10_Conv/FB_FunctionList.TcPOU $ 
* ------------------------------------------------------------------------------------ 
* 	© Swisslog AG 
* 	Swisslog is not liable for any usage of this source code that is not agreed 
* 	on between Swisslog and the other party. The mandatory legal liability remains 
* 	unaffected. 
* ------------------------------------------------------------------------------------ 
* 	Revision History: 
* 
* 	VERSION 		DATE 			INITIALS 			DESCRIPTION 
* 	0.1 			30.11.2018 		mbo					First implementation
* 
**************************************************************************************)
VAR_INPUT
	Execute					: BOOL; // Rising edge triggers new search
	ObservationPosition		: UDINT; // Observation point [mm]
	Range					: UDINT; // Observation point +- Range defines area [mm]
	iWindowTracking			: I_WindowTracking; // Window tracking instance
END_VAR
VAR_OUTPUT
	TrackingZones			: ARRAY[1..MAX_ZONES] OF ST_TrackingZoneInfo; // Found tracking zones
	ZoneCounter 			: INT; // Found zones
	Error					: BOOL; // Configuration error
END_VAR
VAR
	Idx 					: INT; // Iterator
	TrackingZoneIndex		: UINT; // Found tracking zones
	fbTrig					: R_Trig; // Rising edge detection
	StartPosition			: UDINT; // Start search position
	EndPosition 			: UDINT; // End search position
	PositionDelta 			: DINT; // Delta zo zone begin
END_VAR
VAR CONSTANT
	MAX_ZONES				: INT := 5; // Max zones
END_VAR


fbTrig(CLK := Execute);

IF fbTrig.Q THEN
	// Check inputs
	IF iWindowTracking = 0 THEN
		Error := TRUE;
		RETURN;
	END_IF
	
	// Initialize
	Error := FALSE;
	StartPosition := ObservationPosition + Range;
	EndPosition := ObservationPosition - Range;
	ZoneCounter := 0;
	MEMSET(ADR(TrackingZones), 0, SIZEOF(TrackingZones));
	
	FOR Idx := 1 TO MAX_ZONES DO
		
		TrackingZoneIndex := iWindowTracking.M_GetFirstZoneIndex(
								mAbsoluteStartPosition := StartPosition,
								mAbsoluteEndPosition := EndPosition,
								mOnlyZonesWithTU := FALSE);
						
		IF TrackingZoneIndex > 0 THEN
			ZoneCounter := ZoneCounter + 1;
			
			IF ZoneCounter <= MAX_ZONES THEN
			
				PositionDelta := iWindowTracking.M_GetDistanceToZoneStart(ObservationPosition, TrackingZoneIndex);
				
				TrackingZones[ZoneCounter].ZoneIndex := TrackingZoneIndex;
				TrackingZones[ZoneCounter].PositionDelta := PositionDelta;
				TrackingZones[ZoneCounter].ZoneLength := iWindowTracking.P_ZoneTable[TrackingZoneIndex].ZoneLength;
			
				// Update next startposition to limit range
				StartPosition := EndPosition + 1;
			ELSE
				EXIT;
			END_IF
		// Otherwise no zone found, abort search
		ELSE
			EXIT;
		END_IF
	END_FOR
END_IF

END_FUNCTION_BLOCK

// ---- 20_Product/30_Toolbox/99_Misc/13_Helper/FB_MeasureEncoderResolution.TcPOU
/// Uses two defined signals to determine encoder resolution
/// Remark: A constant speed is required for the movement between the signals, to get an accurat result
/// Remark: Drive direction has to be according order of Signal 1 and Signal 2
FUNCTION_BLOCK FB_MeasureEncoderResolution  
(************************************************************************************** 
* 	Application 		: BoxControl Framework 
* 	Revision 			: $Revision: 408723 $ 
* 	Revision date 		: $Date: 2018-06-27 13:49:08 +0200 (Wed, 27 Jun 2018) $ 
* 	Last changed by 	: $Author: b7bolm $ 
* 	URL 				: $URL: http://almscdc.swisslog.com/repo/SWPD/Development/BoxControlFramework/21_Projects/BCF_2.0/trunk/BCF/BCF/JumpStart/20_Product/10_App/12_E_Functions/10_Lib/10_Conv/FB_FunctionList.TcPOU $ 
* ------------------------------------------------------------------------------------ 
* 	© Swisslog AG 
* 	Swisslog is not liable for any usage of this source code that is not agreed 
* 	on between Swisslog and the other party. The mandatory legal liability remains 
* 	unaffected. 
* ------------------------------------------------------------------------------------ 
* 	Revision History: 
* 
* 	VERSION 		DATE 			INITIALS 			DESCRIPTION 
* 	0.1 			22.08.2018 		ale					First implementation
*	0.2				21.09.2018		mbo					Moved and adjusted for standard
* 
**************************************************************************************)
VAR_INPUT
	Run						: BOOL; // Rising edge starts measurement and resets outputs
	StartSignal				: BOOL; // Start measurement
	EndSignal				: BOOL; // Stop measurement
	DistanceSignals			: UINT; // Distance between start and end signal [mm]
	EncoderValueInc			: UDINT; // Encoder values [increment]
	EncoderFW_Desc			: BOOL := FALSE; // Encoder counts in descending sequence 9,8,7,6... to move forward
	MaxEncoderValueInc		: UDINT; // Max value of input "EncoderValue" Remark: Used to detect overflow, needs to be less than DINT size [increment]
END_VAR

VAR_OUTPUT
	Busy					: BOOL; // Measurement running
	DistanceInc				: UDINT; // Distance in increments meausered between the two sensors.
	Resolution				: REAL; // Encoder resolution in increment per milimeter [inc/mm]
	Error					: BOOL; // Overflow during measurement or input value error
END_VAR

VAR
	DeltaEncoderValue		: DINT; // Delta encoder value 
	TrackingEncoderValue	: UDINT; // Internal encoder of traveled increments [increment]
	RunTrig					: R_TRIG; // Run trigger to start measurement and reset
	StartMeasurementTrig	: R_TRIG; // Start signal for measurement
	EndMeasurementTrig		: R_TRIG; // End of measurement
	LastEncoderValueInc		: UDINT; // Last encoder value [increment]
	LastTrackingEncoderValue: UDINT; // Last tracking encoder value [increment]
	StartPosition			: UDINT; // Startposition in increments [increment]
	EndPosition				: UDINT; // Endposition in increments [increment]
END_VAR

// Start measurment and initialize values
RunTrig(clk := Run);

IF RunTrig.Q THEN
	DistanceInc := 0;
	Resolution := 0;
	StartPosition := 0;
	EndPosition := 0;
	DeltaEncoderValue := 0;
	TrackingEncoderValue := 0;
	LastTrackingEncoderValue := 0;
	
	// Check inputs
	IF DistanceSignals = 0 THEN
		Error := TRUE;
	ELSE
		Busy := TRUE;
		Error := FALSE;
	END_IF
END_IF

// When measurement is running, wait for start and end signal
IF Busy AND Run THEN
	// Create internal encoder to make movement independent from encoder overflow
	DeltaEncoderValue := UDINT_TO_DINT(EncoderValueInc) - UDINT_TO_DINT(LastEncoderValueInc);
	
	IF ABS(DeltaEncoderValue) > (UDINT_TO_DINT(MaxEncoderValueInc)/2) THEN
		// Correction with + 1 is to include the 0 in MaxEncoderValue
		IF DeltaEncoderValue < 0 THEN
			DeltaEncoderValue := DeltaEncoderValue + UDINT_TO_DINT(MaxEncoderValueInc) + 1;
		ELSE
			DeltaEncoderValue := UDINT_TO_DINT(EncoderValueInc) - (UDINT_TO_DINT(LastEncoderValueInc) + UDINT_TO_DINT(MaxEncoderValueInc)) - 1;
		END_IF
	END_IF
	
	IF EncoderFW_Desc THEN
		TrackingEncoderValue := DINT_TO_UDINT(UDINT_TO_DINT(TrackingEncoderValue) - DeltaEncoderValue);
	ELSE
		TrackingEncoderValue := DINT_TO_UDINT(UDINT_TO_DINT(TrackingEncoderValue) + DeltaEncoderValue);
	END_IF
	
	// Internal overflow, error
	IF TrackingEncoderValue < LastTrackingEncoderValue THEN
		Error := TRUE;
		Busy := FALSE;
		RETURN;
	END_IF

	LastEncoderValueInc := EncoderValueInc;
	LastTrackingEncoderValue := TrackingEncoderValue;

	// Wait for front edge
	StartMeasurementTrig(clk := StartSignal);
	
	IF StartMeasurementTrig.Q THEN
		StartPosition := TrackingEncoderValue;
	END_IF
	
	// Wait for rear edge
	EndMeasurementTrig(clk := EndSignal);
	
	IF EndMeasurementTrig.Q THEN
		EndPosition := TrackingEncoderValue;
		
		IF EndPosition >= StartPosition THEN
			DistanceInc := EndPosition - StartPosition;
			Resolution := UDINT_TO_REAL(DistanceInc) / UINT_TO_REAL(DistanceSignals);
		// Otherwise overflow, distance greather than data type UDINT 
		ELSE
			Error := TRUE;
		END_IF
		
		Busy := FALSE;
	END_IF
ELSIF Busy THEN
	Busy := FALSE;
	Error := TRUE;
END_IF

END_FUNCTION_BLOCK

// ---- 20_Product/30_Toolbox/99_Misc/13_Helper/FB_ScaleEncoder.TcPOU
/// This function block scales an encoder increments to milimeter and aligns counting direction (EncoderFwDesc)
FUNCTION_BLOCK FB_ScaleEncoder
(************************************************************************************** 
* 	Application 		: BoxControl Framework 
* 	Revision 			: $Revision: 408723 $ 
* 	Revision date 		: $Date: 2018-06-27 13:49:08 +0200 (Wed, 27 Jun 2018) $ 
* 	Last changed by 	: $Author: b7bolm $ 
* 	URL 				: $URL: http://almscdc.swisslog.com/repo/SWPD/Development/BoxControlFramework/21_Projects/BCF_2.0/trunk/BCF/BCF/JumpStart/20_Product/10_App/12_E_Functions/10_Lib/10_Conv/FB_FunctionList.TcPOU $ 
* ------------------------------------------------------------------------------------ 
* 	© Swisslog AG 
* 	Swisslog is not liable for any usage of this source code that is not agreed 
* 	on between Swisslog and the other party. The mandatory legal liability remains 
* 	unaffected. 
* ------------------------------------------------------------------------------------ 
* 	Revision History: 
* 
* 	VERSION 		DATE 			INITIALS 			DESCRIPTION 
* 	0.1 			25.09.2018 		mbo					First implementation
* 
**************************************************************************************)
VAR_INPUT
	EncoderValueInc			: UDINT; // Encoder value [increment]
	MaxEncoderValueInc		: UDINT; // Max encoder value (Range is 0..MaxValue) [increment]
	IncrementPerMM			: LREAL; // Increment per milimeter [inc/mm]
END_VAR
VAR_OUTPUT
	ScaledEncoderValue		: UDINT; // Scaled encoder signal [mm] (Delta + = fwd)
	ScaledMaxEncoderValue	: UDINT; // Scaled max encoder value [mm]
	Error					: BOOL; // Input error 
END_VAR
VAR
	ScaledEncoderValueReal 	: LREAL; // Scaled encoder value as real value
END_VAR

// Init
ScaledEncoderValue := 0;

// Validate inputs
IF IncrementPerMM = 0 OR 
   MaxEncoderValueInc = 0 THEN
	Error := TRUE;
	RETURN;
END_IF

Error := FALSE;

// Update max scaled encoder value (Trunc is used to truncate decimal places and not do auto rounding)
ScaledMaxEncoderValue := LREAL_TO_UDINT(LTRUNC(UDINT_TO_LREAL(MaxEncoderValueInc) / IncrementPerMM));

// Convert pulses into pulses per mm
ScaledEncoderValueReal := UDINT_TO_LREAL(EncoderValueInc) / IncrementPerMM;

// truncate decimal places (e.g. 5,3 -> 5 ; -3,2  -> -3)
ScaledEncoderValue := LREAL_TO_UDINT(LTRUNC(ScaledEncoderValueReal));

END_FUNCTION_BLOCK

// ---- 20_Product/30_Toolbox/99_Misc/13_Helper/FB_Throughput.TcPOU
FUNCTION_BLOCK FB_Throughput
(**************************************************************************************
 * 	Application		:	BoxControl Framework
 *	Revision		:	$Revision: 453140 $
 *	Revision date	:	$Date: 2020-05-28 08:47:05 +0200 (tor, 28 maj 2020) $
 *	Last changed by	:	$Author: b7muotj $
 *	URL				:	$URL: http://almscdc.swisslog.com/repo/SWPD/Development/BoxControlFramework/20_Release/tags/R1.12.0/01_Software/BCF/BCF/JumpStart/30_Toolbox/99_Misc/13_Helper/FB_Throughput.TcPOU $
 *
 *	Purpose			:	The Function block calculates two throughput values "Throughput" and "ThroughputLongTerm" that are normalised to TU's per Hour [TU/h].
 *
 * ------------------------------------------------------------------------------------
 *	Copyright Swisslog [IP AG], Switzerland. All rights reserved.
 * 
 * ------------------------------------------------------------------------------------
 *	
 * 	Revision History: 
 *
 * 	VERSION			DATE			INITIALS			DESCRIPTION
 *	0.1				01.01.2015		ahe					Example
 *	0.2				19.05.2020		jmu					Comments added, cleaned, added check for division 0. Added to the BCF
 *
 **************************************************************************************)
VAR_INPUT
	eFunctionNumber			: E_FunctionNumber; //FunctionNumber whose throughput is being measured
	ZoneIndex				: INT; //Index of zone whose throughput is being measured in the given function
	TimeInterval			: TIME; //Update time interval of the output Throughput 
	TimeIntervalLongTerm	: TIME; //Update time interval of the output ThroughputLongTerm
END_VAR
VAR_OUTPUT
	Throughput				: INT; //Output updated on intervals defined by TimeInterval normalised to TU/h
	ThroughputLongTerm		: INT; //Output updated ont intervals defined by TimeIntervalLongTerm normalised to TU/h
END_VAR
VAR
	ZoneData				: ST_TransportControlData;
	LastSensorOccoupied		: BOOL;
	TU_Counter				: UDINT;
	TU_CounterLongTerm		: UDINT;
	TU_CounterOverall		: UDINT;
	fbTimer					: FB_Timer;
	fbTimerLongTerm			: FB_Timer;
END_VAR

IF ZoneIndex > 0 AND ZoneIndex <= NUMBER_OF_ZONES_PER_FUNCTION
   AND eFunctionNumber > E_FunctionNumber.F_BEGIN_FUNCTION
   AND eFunctionNumber < E_FunctionNumber.F_END_FUNCTION THEN
   
	ZoneData := F_GetTransportControlData(eFunctionNumber, ZoneIndex);

	//Count up on positive edge	
	IF ZoneData.SensorOccupied AND NOT LastSensorOccoupied THEN
		TU_Counter := TU_Counter + 1;
		TU_CounterLongTerm := TU_CounterLongTerm + 1;
		TU_CounterOverall := TU_CounterOverall + 1;
	END_IF

	LastSensorOccoupied := ZoneData.SensorOccupied;

	//Calculate outputs after each period has passed	
	fbTimer(IN := TRUE, PT := TimeInterval);
	fbTimerLongTerm(IN := TRUE, PT := TimeIntervalLongTerm);

	IF fbTimer.Q THEN
		IF TimeInterval <> T#0S THEN
			Throughput := UDINT_TO_INT(TIME_TO_UDINT(T#1H) / TIME_TO_UDINT(TimeInterval) * TU_Counter);
		ELSE
			Throughput := 0;
		END_IF	
			TU_Counter := 0;
			fbTimer(IN := FALSE);		
	END_IF
	
	IF fbTimerLongTerm.Q THEN
		IF TimeIntervalLongTerm <> T#0S THEN		
			ThroughputLongTerm := UDINT_TO_INT(TIME_TO_UDINT(T#1H) / TIME_TO_UDINT(TimeIntervalLongTerm) * TU_CounterLongTerm);
		ELSE		
			ThroughputLongTerm := 0;
		END_IF
		TU_CounterLongTerm := 0;
		fbTimerLongTerm(IN := FALSE);
	END_IF

END_IF

END_FUNCTION_BLOCK

// ---- 20_Product/30_Toolbox/99_Misc/13_Helper/FB_TrackingReservation.TcPOU
/// This function block automatically reserves a zone on the window tracking.
/// Remark: Only one zone at the time
FUNCTION_BLOCK FB_TrackingReservation IMPLEMENTS I_TrackingActionListener
(************************************************************************************** 
* 	Application 		: BoxControl Framework 
* 	Revision 			: $Revision: 408723 $ 
* 	Revision date 		: $Date: 2018-06-27 13:49:08 +0200 (Wed, 27 Jun 2018) $ 
* 	Last changed by 	: $Author: b7bolm $ 
* 	URL 				: $URL: http://almscdc.swisslog.com/repo/SWPD/Development/BoxControlFramework/21_Projects/BCF_2.0/trunk/BCF/BCF/JumpStart/20_Product/10_App/12_E_Functions/10_Lib/10_Conv/FB_FunctionList.TcPOU $ 
* ------------------------------------------------------------------------------------ 
* 	© Swisslog AG 
* 	Swisslog is not liable for any usage of this source code that is not agreed 
* 	on between Swisslog and the other party. The mandatory legal liability remains 
* 	unaffected. 
* ------------------------------------------------------------------------------------ 
* 	Revision History: 
* 
* 	VERSION 		DATE 			INITIALS 			DESCRIPTION 
* 	0.1 			25.09.2018 		mbo					First implementation
* 
**************************************************************************************)
VAR_INPUT
	Enable					: BOOL; // Enable reservation
	ActionId				: INT; // Action id for zone
	AbsolutePosition		: DINT; // Position where it should be earliest reserved
	Length					: UINT; // length of tracking zone to be reserved
	MaxDistance				: UDINT; // Max distance in which its allowed to be reserved (0=Full range)
	PositionToLive			: UDINT; // Position after the reserved zones gets deleted if not used
	MinimumDistance			: UINT; // Minimum gap until next reservation [mm]
	iWindowTracking			: I_WindowTracking; // Link to window tracking
END_VAR
VAR_OUTPUT
	ReservedZoneIndex		: UINT; // Currently reserved zone index
END_VAR
VAR
	LastReservedZoneIndex	: UINT; // Last reserved zone index
	LastZoneEndPosition		: UDINT; // Last zone end position
END_VAR

// Check inputs
IF iWindowTracking = 0 OR 
   ActionId = 0 OR
   Length = 0 THEN
	RETURN;
END_IF

// Reserve a new zone if required
IF Enable THEN
	
	IF ReservedZoneIndex = 0 THEN
		LastZoneEndPosition := iWindowTracking.M_GetZoneEndPosition(LastReservedZoneIndex);
		
		IF AbsolutePosition + MinimumDistance < UDINT_TO_DINT(LastZoneEndPosition) OR LastZoneEndPosition = 0 THEN
			ReservedZoneIndex := iWindowTracking.M_AllocateNextFreeZone(
													mActionId 			:= ActionId,
													mAbsolutePosition 	:= DINT_TO_UDINT(AbsolutePosition),
													mLength 			:= Length,
													mMaxDistance 		:= MaxDistance,
													miActionListener 	:= THIS^,
													mPositionToLive 	:= PositionToLive);
		END_IF
	END_IF
END_IF

METHOD M_ActionZoneChangedEvent

VAR_INPUT
	mZoneIndex	: UINT; // Deleted zone index
	mZoneData	: ST_WindowTrackingZone; // Data of deleted zone
END_VAR
// Reset when zone gets occupied
IF mZoneData.TU_Present THEN
	LastReservedZoneIndex := ReservedZoneIndex;
	ReservedZoneIndex := 0;
END_IF
END_METHOD

// Automatically called whenever the stored zone gets deleted on tracking
METHOD M_ActionZoneDeletedEvent
VAR_INPUT
	mZoneIndex	: UINT; //  Deleted zone index
	mZoneData	: ST_WindowTrackingZone; // Data of deleted zone
END_VAR
IF mZoneIndex = ReservedZoneIndex THEN
	ReservedZoneIndex := 0;
	
ELSIF mZoneIndex = LastReservedZoneIndex THEN
	LastReservedZoneIndex := 0;
END_IF
END_METHOD

/// Delete pending reservation
METHOD M_ClearReservation : BOOL // Returns true if successfully deleted
VAR_INPUT
END_VAR
M_ClearReservation := FALSE;

IF iWindowTracking <> 0 THEN
	IF ReservedZoneIndex > 0 THEN
		M_ClearReservation := iWindowTracking.M_DeleteZone(ReservedZoneIndex);
	END_IF
END_IF
END_METHOD

END_FUNCTION_BLOCK

// ---- 20_Product/30_Toolbox/99_Misc/13_Helper/F_AlignEncoderValue.TcPOU
FUNCTION F_AlignEncoderValue : UDINT
(************************************************************************************** 
* 	Application 		: BoxControl Framework 
* 	Revision 			: $Revision: 408723 $ 
* 	Revision date 		: $Date: 2018-06-27 13:49:08 +0200 (Wed, 27 Jun 2018) $ 
* 	Last changed by 	: $Author: b7bolm $ 
* 	URL 				: $URL: http://almscdc.swisslog.com/repo/SWPD/Development/BoxControlFramework/21_Projects/BCF_2.0/trunk/BCF/BCF/JumpStart/20_Product/10_App/12_E_Functions/10_Lib/10_Conv/FB_FunctionList.TcPOU $ 
* ------------------------------------------------------------------------------------ 
* 	© Swisslog AG 
* 	Swisslog is not liable for any usage of this source code that is not agreed 
* 	on between Swisslog and the other party. The mandatory legal liability remains 
* 	unaffected. 
* ------------------------------------------------------------------------------------ 
* 	Revision History: 
* 
* 	VERSION 		DATE 			INITIALS 			DESCRIPTION 
* 	0.1 			25.09.2018 		mbo					First implementation
* 
**************************************************************************************)
VAR_INPUT
	EncoderValueInc				: UDINT; // Encoder value [increment]
	MaxEncoderValueInc			: UDINT; // Max encoder value (Range is 0..MaxValue) [increment]
	EncoderFW_Desc				: BOOL := FALSE; // Encoder counts in descending sequence 9,8,7,6... to move forward
END_VAR


IF EncoderValueInc = 0 THEN
	F_AlignEncoderValue := 0;
	RETURN;
END_IF

IF EncoderFW_Desc THEN
	// In:   0 5 4 3 2 1 0 5 4 3 2 1
	// Out:  0 1 2 3 4 5 0 1 2 3 4 5
	// Remark: 0 = 0, this is important otherwise a step would be detected
	// on system startup. 
	F_AlignEncoderValue := MaxEncoderValueInc - EncoderValueInc + 1;
ELSE
	// In:    0 1 2 3 4 5 0 1 2 3 4 5
	// Out:	  0 1 2 3 4 5 0 1 2 3 4 5
	F_AlignEncoderValue := EncoderValueInc;
END_IF

END_FUNCTION

// ---- 20_Product/30_Toolbox/99_Misc/13_Helper/F_CountTUs.TcPOU
FUNCTION F_CountTUs : INT
(**************************************************************************************
 * 	Application		:	BoxControl Framework
 *	Revision		:	$Revision: 453155 $
 *	Revision date	:	$Date: 2020-05-28 10:31:40 +0200 (tor, 28 maj 2020) $
 *	Last changed by	:	$Author: b7muotj $
 *	URL				:	$URL: http://almscdc.swisslog.com/repo/SWPD/Development/BoxControlFramework/20_Release/tags/R1.12.0/01_Software/BCF/BCF/JumpStart/30_Toolbox/99_Misc/13_Helper/F_CountTUs.TcPOU $
 *
 *	Purpose			:	Counts present TU's on Function range between BeginCount and EndCount
 *
 * ------------------------------------------------------------------------------------
 *	Copyright Swisslog [IP AG], Switzerland. All rights reserved.
 * 
 * ------------------------------------------------------------------------------------
 *	
 * 	Revision History: 
 *
 * 	VERSION			DATE			INITIALS			DESCRIPTION
 *	0.1				27.05.2020		jmu					Added to the BCF
 *
 **************************************************************************************)
VAR_INPUT
	BeginCount	: E_FunctionNumber; // Function to start the counting of TU's
	EndCount	: E_FunctionNumber; // Function to stop the counting of TU's
END_VAR
VAR
	eFunctionNumber	: E_FunctionNumber;
	i	: INT;
END_VAR

F_CountTUs := 0;

//Look for the count of present TUs within the range and add found TUs together
IF EndCount >= BeginCount 
	AND BeginCount > F_BEGIN_FUNCTION 
	AND EndCount < F_END_FUNCTION THEN
	
	FOR eFunctionNumber := BeginCount TO EndCount DO
		
		IF FunctionRegistry[eFunctionNumber].Enable THEN
			
			IF __ISVALIDREF(FunctionRegistry[eFunctionNumber].rFunction) THEN
				
				FOR i := 1 TO NUMBER_OF_ZONES_PER_FUNCTION DO
					
					F_CountTUs:=F_CountTUs + UINT_TO_INT(FunctionRegistry[eFunctionNumber].rFunction.ZoneData[i].TransportControlData.NumberOfPresentTUs);
				END_FOR
			END_IF
		END_IF
	END_FOR
END_IF

END_FUNCTION

// ---- 20_Product/30_Toolbox/99_Misc/13_Helper/F_CountTUsWithDestination.TcPOU
FUNCTION F_CountTUsWithDestination : INT
(**************************************************************************************
 * 	Application		:	BoxControl Framework
 *	Revision		:	$Revision: 453155 $
 *	Revision date	:	$Date: 2020-05-28 10:31:40 +0200 (tor, 28 maj 2020) $
 *	Last changed by	:	$Author: b7muotj $
 *	URL				:	$URL: http://almscdc.swisslog.com/repo/SWPD/Development/BoxControlFramework/20_Release/tags/R1.12.0/01_Software/BCF/BCF/JumpStart/30_Toolbox/99_Misc/13_Helper/F_CountTUsWithDestination.TcPOU $
 *
 *	Purpose			:	Counts present TU's on Function range between BeginCount and EndCount with certain destination
 *
 * ------------------------------------------------------------------------------------
 *	Copyright Swisslog [IP AG], Switzerland. All rights reserved.
 * 
 * ------------------------------------------------------------------------------------
 *	
 * 	Revision History: 
 *
 * 	VERSION			DATE			INITIALS			DESCRIPTION
 *	0.1				27.05.2020		jmu					Added to the BCF
 *
 **************************************************************************************)
VAR_INPUT
	BeginCount	: E_FunctionNumber; // Function to start the counting of TU's
	EndCount	: E_FunctionNumber; // Function to stop the counting of TU's
	Destination: E_FunctionNumber; // Destination of TU's to involve in the count
END_VAR
VAR
	eFunctionNumber: E_FunctionNumber;
	rFunction: REFERENCE TO FB_FunctionConv;
	i: INT;
END_VAR

F_CountTUsWithDestination := 0;

//Look for the count of present TUs within the range and add found TUs together if the destination matches the desired one
IF EndCount >= BeginCount 
	AND BeginCount > F_BEGIN_FUNCTION 
	AND EndCount < F_END_FUNCTION THEN
	
	FOR eFunctionNumber := BeginCount TO EndCount DO
		
		IF FunctionRegistry[eFunctionNumber].Enable THEN
			
			IF __ISVALIDREF(FunctionRegistry[eFunctionNumber].rFunction) THEN
				
				rFunction REF= FunctionRegistry[eFunctionNumber].rFunction;
				FOR i := 1 TO NUMBER_OF_ZONES_PER_FUNCTION DO
					
					IF rFunction.zoneData[i].TransportControlData.TU_DataIndex <> 0 
						AND TU_DataTable[rFunction.zoneData[i].TransportControlData.TU_DataIndex].Destination[1].eFunctionNumber = Destination THEN
						
							F_CountTUsWithDestination:=F_CountTUsWithDestination+1;
					END_IF
				END_FOR
			END_IF
		END_IF
	END_FOR
END_IF

END_FUNCTION

// ---- 20_Product/30_Toolbox/99_Misc/FB_Encoder.TcPOU
FUNCTION_BLOCK FB_Encoder
(**************************************************************************************
 * 	Application		:	BoxControl Framework
 *	Revision		:	$Revision: 475083 $
 *	Revision date	:	$Date: 2021-04-10 12:07:10 +0200 (lör, 10 apr 2021) $
 *	Last changed by	:	$Author: d7mangc $
 *	URL				:	$URL: http://almscdc.swisslog.com/repo/SWPD/Development/BoxControlFramework/20_Release/tags/R1.12.0/01_Software/BCF/BCF/JumpStart/30_Toolbox/99_Misc/FB_Encoder.TcPOU $
 *
 *	Purpose			:	Simple encoder
 *
 * ------------------------------------------------------------------------------------
 *	Copyright Swisslog [IP AG], Switzerland. All rights reserved.
 * 
 * ------------------------------------------------------------------------------------
 *	
 * 	Revision History: 
 *
 * 	VERSION			DATE			INITIALS			DESCRIPTION
 *	0.1				01.01.2001		swl					Example
 *
 **************************************************************************************)
VAR_INPUT
	Speed			: REAL		:= 0.0;		// Speed [mm/s]
	Run				: BOOL		:= FALSE;	// Run command
	Resolution		: INT		:= 1;		// Encoder Resolution [Inc/mm]
END_VAR

VAR_OUTPUT
	EncoderValue	: WORD		:= 0;		// Encoder value [Inc]
END_VAR

VAR
	TimeTick		: TIME		:= T#0S;		// Timestamp last calculation
	Position		: LREAL		:= 0;			// Current encoder position
	CalcSpeed		: LREAL		:= 0;			// Current used speed to calculate
	LastSpeed		: LREAL		:= 0;			// Speed from last cycle
	Temp			: LREAL		:= 0;			// Aux value to calculate
	Inc				: LREAL		:= 0;			// Change in increments in this cycle
	CycleTime		: LREAL		:= 0;			// Current cycle time in seconds
END_VAR

// Get current cycle time
CycleTime := TIME_TO_LREAL( F_GetTimeMsDiff(TimeTick) ) / 1_000; // ms -> s
TimeTick  := F_GetTimeMsTick();

// Simulation at standstill -> no counting
IF NOT Run THEN
	CalcSpeed:= 0;
ELSE
	CalcSpeed:= ABS(Speed);
END_IF

// Calculate increment based on speed and resolution
Temp := (CalcSpeed - LastSpeed); 
Temp := (Temp / 2) + CalcSpeed;

LastSpeed := CalcSpeed;

// Update encoder value
Inc      := (Temp * Resolution * CycleTime);
Position := Position + Inc;

// Update output value as word
EncoderValue:= LREAL_TO_WORD(Position); // Cut off at 2^16

END_FUNCTION_BLOCK

// ---- 20_Product/10_BCF/BCF_Version.TcTLO
TEXTLIST BCF_Version
  Version = 'R1.12.0'
  Company = 'Swisslog'
   = ''
END_TEXTLIST

// ---- 20_Product/20_ProBox/40_TC_Visualization/10_Controls/LoopControl/V_LoopControl.TcVIS
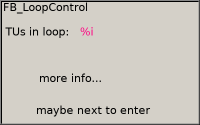
VISUALIZATION V_LoopControl  // 200x125
VAR_IN_OUT
	{attribute 'VAR_IN_OUT_AS_POINTER'}
	fbFunction		: FB_LoopControl;	
END_VAR
    Rectangle (0,0 200x125)
    Label (0,0 200x15), "FB_LoopControl"
    Rectangle (77,22 67x20), "%i", text variable: fbFunction.TuCountInLoop, colour toggle: fbFunction.LoopIsFull
    Label (36,71 92x15), "more info..."
    Label (33,103 123x15), "maybe next to enter"
    Label (4,17 67x30), "TUs in loop:"
END_VISUALIZATION

// ---- 20_Product/20_ProBox/40_TC_Visualization/10_Controls/TransportControl/V_TransportControl.TcVIS
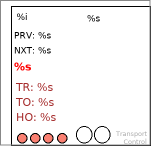
VISUALIZATION V_TransportControl  // 151x146
VAR_IN_OUT	
	{attribute 'VAR_IN_OUT_AS_POINTER'}
	TransportControl	: FB_ProBoxTransportControl;
	ZoneData			: ST_ZoneData;
		
END_VAR
    Rectangle (11,6 140x140), colour toggle: ZoneData.TransportControlData.NumberOfPresentTUs>0
    Rectangle (13,110 130x15), "HO: %s", text variable: ZoneData.TransportControlData.eHandOverState
    Rectangle (13,95 130x15), "TO: %s", text variable: ZoneData.TransportControlData.eTakeOverState
    Rectangle (13,80 130x15), "TR: %s", text variable: ZoneData.TransportControlData.eTransportState
    Rectangle (36,6 115x25), "%s", tooltip "TU ID", text variable: TU_DataTable[ZoneData.TransportControlData.TU_DataIndex].TU_ID.ASCII
    Rectangle (11,28 140x15), "PRV: %s", text variable: TransportControl.PrevTransportData.eFunctionNumber
    Rectangle (11,43 140x15), "NXT: %s", text variable: TransportControl.NextTransportData.eFunctionNumber
    Ellipse (17,133 10x10), tooltip "'Indicator shows that addon(s) is available -> Enable signal'", colour toggle: ZoneData.AddOn.Orders.Enable, invisible if: ZoneData.AddOn.NoAddons
    Ellipse (30,133 10x10), tooltip "'Indicator shows that addon(s) is available - Enable Takeover'", colour toggle: ZoneData.AddOn.Orders.EnableTakeover, invisible if: ZoneData.AddOn.NoAddons
    Ellipse (43,133 10x10), tooltip "'Indicator shows that addon(s) is available - Enable Handover'", colour toggle: ZoneData.AddOn.Orders.EnableHandover, invisible if: ZoneData.AddOn.NoAddons
    Ellipse (57,133 10x10), tooltip "'Indicator shows that addon(s) is available - Data Ready'", colour toggle: ZoneData.AddOn.Orders.DataReady, invisible if: ZoneData.AddOn.NoAddons
    Ellipse (94,126 16x17), tooltip "sensor occupied", colour toggle: ZoneData.TransportControlData.SensorOccupied
    Label (102,130 48x16), "Transport Control"
    Rectangle (11,57 140x20), "%s", tooltip "%s", text variable: ZoneData.ErrorData.Error.ErrorCode.Conv, invisible if: ZoneData.ErrorData.Error.ErrorCode.Conv = 0
        p4168582468: ZoneData.ErrorData.Error.ErrorParam
    Rectangle (11,6 22x22), "%i", tooltip "TU index", text variable: ZoneData.TransportControlData.TU_DataIndex
    Ellipse (76,126 16x17), tooltip "Transportcontrol Occupied", colour toggle: ZoneData.TransportControlData.Occupied
END_VISUALIZATION

// ---- 20_Product/20_ProBox/40_TC_Visualization/11_Addon/CraneXoverAddon/V_CraneXoverAddon.TcVIS
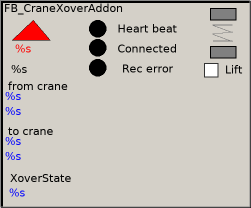
VISUALIZATION V_CraneXoverAddon  // 251x208
VAR_IN_OUT
	{attribute 'VAR_IN_OUT_AS_POINTER'}
	fbFunction		: FB_CraneXoverAddon;	

END_VAR
    Rectangle (1,1 250x207)
    Label (1,1 200x15), "FB_CraneXoverAddon"
    Rectangle (12,39 70x20), "%s", text variable: fbFunction.ZoneData[1].ErrorData.Error.ErrorCode.Conv, invisible if: fbFunction.FunctionData.ErrorData.Error.ErrorCode.Conv = 0
    Polygon (12,40) (33,20) (50,40) (44,40) (22,40), invisible if: fbFunction.FunctionData.ErrorData.ErrorState = E_ErrorState.OPERATIONAL
    Rectangle (6,183 239x20), "%s", tooltip "XoverState", text variable: fbFunction._XoverState
    Rectangle (2,149 248x15), "%s", text variable: fbFunction.HW_Outputs.HandshakeCraneInterfaceSend.HandOverState
    Rectangle (2,134 246x15), "%s", text variable: fbFunction.HW_Outputs.HandshakeCraneInterfaceSend.TakeOverState
    Label (5,124 124x15), "to crane"
    Rectangle (2,89 245x15), "%s", text variable: fbFunction.Inputs.HandshakeCraneInterfaceReceive.TakeOverState
    Rectangle (2,104 246x15), "%s", text variable: fbFunction.Inputs.HandshakeCraneInterfaceReceive.HandOverState
    Label (5,79 124x15), "from crane"
    Rectangle (210,8 26x12), tooltip "Upper lift sensor", colour toggle: fbFunction.HW_Inputs.Sensor_Pos_Up
    Rectangle (210,46 26x12), tooltip "Lower lift sensor", colour toggle: fbFunction.HW_Inputs.Sensor_Pos_Down
    Polyline (232,25) (213,25) (232,32) (213,34) (232,41) (213,41), colour toggle: fbFunction.HW_Outputs.Drive_Run_UpDown
    Label (7,171 124x15), "XoverState"
    Checkbox (202,60 49x20), "Lift", variable: fbFunction.Settings.LiftEnabled, input disabled if: TRUE
    Ellipse (89,20 17x17), colour toggle: fbFunction.HW_Inputs.HandshakeCraneInterfaceReceive.Watchdog
    Label (109,21 77x16), "Heart beat"
    Ellipse (89,39 17x17), colour toggle: fbFunction._fbCranePlcTcpcom.Connected
    Ellipse (89,59 17x17), colour toggle: fbFunction._fbCranePlcTcpcom.ReceiveDataError
    Label (109,41 77x16), "Connected"
    Label (109,61 77x16), "Rec error"
    Rectangle (8,62 76x15), "%s", text variable: fbFunction._fbCranePlcTcpcom.Config.RemotePort
END_VISUALIZATION

// ---- 20_Product/20_ProBox/40_TC_Visualization/11_Addon/FastDoorAddon/V_FastDoorAddon.TcVIS
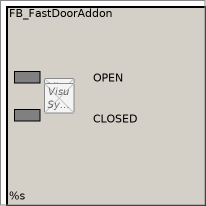
VISUALIZATION V_FastDoorAddon  // 206x206
VAR_IN_OUT
	fbFunction 	: FB_FastDoorAddon;
END_VAR
    Rectangle (6,6 200x200)
    Rectangle (6,186 200x20), "%s", text variable: fbFunction.ConfigFunction.FunctionName
    Label (6,6 200x15), "FB_FastDoorAddon"
    Rectangle (14,109 26x12), tooltip "Door lift sensor", colour toggle: fbFunction.HW_Inputs.Closed
    Rectangle (14,71 26x12), tooltip "Door up sensor", colour toggle: fbFunction.HW_Inputs.Open
    Image (44,78 30x30), tooltip "Door moving up", invisible if: NOT fbFunction.HW_Outputs.OpenDoor, image: VisuSymbols.Symbols.ArrowBoldUp
    Image (44,83 30x30), tooltip "Door moving down", invisible if: NOT fbFunction.HW_Outputs.CloseDoor, image: VisuSymbols.Symbols.ArrowBoldDown
    Rectangle (90,68 60x20), "OPEN", tooltip "Door open", text variable: fbFunction.ConfigFunction.FunctionName, invisible if: NOT fbFunction.HW_Inputs.Open
    Rectangle (90,109 60x20), "CLOSED", tooltip "Door closed", text variable: fbFunction.ConfigFunction.FunctionName, invisible if: NOT fbFunction.HW_Inputs.Closed
END_VISUALIZATION

// ---- 20_Product/20_ProBox/40_TC_Visualization/11_Addon/InOutFeedAddon/V_InOutFeedAddon.TcVIS
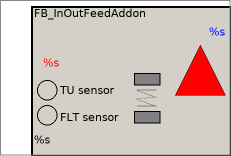
VISUALIZATION V_InOutFeedAddon  // 231x156
VAR_IN_OUT
	{attribute 'VAR_IN_OUT_AS_POINTER'}
	fbFunction		: FB_InOutFeedAddon;	
END_VAR
    Rectangle (31,6 200x150)
    Label (31,6 199x15), "FB_InOutFeedAddon"
    Rectangle (31,130 199x20), "%s", text variable: fbFunction.ConfigFunction.FunctionName
    Rectangle (40,53 160x20), "%s", text variable: fbFunction.ZoneData[1].ErrorData.Error.ErrorCode.Conv, invisible if: fbFunction.FunctionData.ErrorData.Error.ErrorCode.Conv = 0
    Polygon (175,95) (200,45) (225,95) (210,95) (190,95), invisible if: fbFunction.FunctionData.ErrorData.ErrorState = E_ErrorState.OPERATIONAL
    Rectangle (68,22 160x20), "%s", text variable: fbFunction.InOutFeedState.eState
    Ellipse (37,80 20x20), colour toggle: fbFunction.Inputs.HW.TUSensor
    Label (57,83 92x15), "TU sensor"
    Ellipse (37,105 20x20), colour toggle: fbFunction.Inputs.HW.FLTSensor
    Label (57,110 92x15), "FLT sensor"
    Polyline (156,90) (137,90) (156,97) (137,99) (156,106) (137,106), colour toggle: fbFunction.HW_Outputs.Drive_Run_UpDown, invisible if: NOT fbFunction.Settings.LiftEnabled
    Rectangle (134,111 26x12), tooltip "Lower lift sensor", colour toggle: fbFunction.HW_Inputs.Sensor_Pos_Down, invisible if: NOT fbFunction.Settings.LiftEnabled
    Rectangle (134,73 26x12), tooltip "Upper lift sensor", colour toggle: fbFunction.HW_Inputs.Sensor_Pos_Up, invisible if: NOT fbFunction.Settings.LiftEnabled
END_VISUALIZATION

// ---- 20_Product/20_ProBox/40_TC_Visualization/11_Addon/LiftTableAddon/V_LiftTableAddon.TcVIS
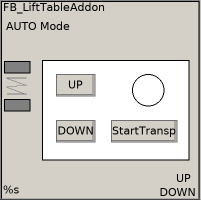
VISUALIZATION V_LiftTableAddon  // 201x200
VAR_IN_OUT
	{attribute 'VAR_IN_OUT_AS_POINTER'}
	fbFunction 		: FB_LiftTableAddon;
	fbEmuFunction	: FB_LiftTableAddonEmulation;
END_VAR
    Rectangle (0,0 200x200), colour toggle: fbFunction.HW_Outputs.LiftDown OR fbFunction.HW_Outputs.LiftUp
    Rectangle (0,180 200x20), "%s", text variable: fbFunction.ConfigFunction.FunctionName
    Label (0,0 200x15), "FB_LiftTableAddon"
    Label (166,172 35x13), "UP", invisible if: NOT fbFunction.HW_Outputs.LiftUp
    Label (155,185 45x15), "DOWN", invisible if: NOT fbFunction.HW_Outputs.LiftDown
    Polyline (26,78) (7,78) (26,85) (7,87) (26,94) (7,94), colour toggle: fbFunction.HW_Outputs.LiftUp OR fbFunction.HW_Outputs.LiftDown
    Rectangle (4,99 26x12), tooltip "Lower lift sensor", colour toggle: fbFunction.HW_Inputs.Lift.SensorPosDown
    Rectangle (4,61 26x12), tooltip "Upper lift sensor", colour toggle: fbFunction.HW_Inputs.Lift.SensorPosUp
    RoundedRectangle (42,60 147x100)
    Button (56,120 39x22), "DOWN"
        tap fbEmuFunction.DebugOpDown
    Button (111,120 66x22), "StartTransp"
        tap fbEmuFunction.DebugOpStartTransp
    Ellipse (132,74 32x32), colour toggle: fbFunction.HW_Outputs.StartTransport
    Button (56,74 39x22), "UP"
        tap fbEmuFunction.DebugOpUp
    Label (3,20 79x13), "AUTO Mode", invisible if: fbFunction.Settings.OperatorPanelEnable
END_VISUALIZATION

// ---- 20_Product/20_ProBox/40_TC_Visualization/11_Addon/PalletCheckAddon/V_PalletCheckAddon.TcVIS
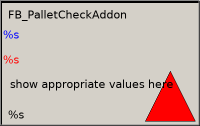
VISUALIZATION V_PalletCheckAddon  // 200x126
VAR_IN_OUT
	{attribute 'VAR_IN_OUT_AS_POINTER'}
	fbFunction		: FB_PalletCheckAddon;
END_VAR
    Rectangle (0,1 200x125)
    Rectangle (5,105 143x20), "%s", text variable: fbFunction.ConfigFunction.FunctionName
    Label (5,5 158x20), "FB_PalletCheckAddon"
    Rectangle (0,25 99x20), "%s", text variable: fbFunction.eState
    Polygon (145,121) (170,71) (195,121) (180,121) (160,121), invisible if: fbFunction.FunctionData.ErrorData.ErrorState = E_ErrorState.OPERATIONAL
    Rectangle (0,50 161x20), "%s", text variable: fbFunction.FunctionData.ErrorData.Error.ErrorCode.Conv, invisible if: fbFunction.FunctionData.ErrorData.Error.ErrorCode.Conv = 0
    Label (7,77 158x15), "show appropriate values here"
END_VISUALIZATION

// ---- 20_Product/20_ProBox/40_TC_Visualization/11_Addon/PalletMagazineAddon/V_PalletMagazineAddon.TcVIS
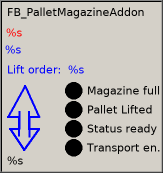
VISUALIZATION V_PalletMagazineAddon  // 163x173
VAR_IN_OUT
	{attribute 'VAR_IN_OUT_AS_POINTER'}
	fbFunction		: FB_PalletMagazineAddon;	
END_VAR
    Rectangle (0,0 163x173)
    Label (4,5 146x15), "FB_PalletMagazineAddon"
    Rectangle (4,151 104x20), "%s", text variable: fbFunction.ConfigFunction.FunctionName
    Rectangle (3,23 157x20), "%s", tooltip "%s", text variable: fbFunction.FunctionData.ErrorData.Error.ErrorCode.Conv, invisible if: fbFunction.FunctionData.ErrorData.Error.ErrorCode.Conv = 0
        p4168582468: fbFunction.FunctionData.ErrorData.Error.ErrorParam
    Rectangle (2,40 161x20), "%s", text variable: fbFunction.BaseFunctionData.States.eState
    Rectangle (4,60 155x20), "Lift order: %s", text variable: fbFunction.BaseFunctionData.OrderPosLift
    Polyline (19,136) (19,117) (8,117) (25,86) (39,117) (29,117) (29,137), invisible if: NOT fbFunction.HW_Outputs.LiftUp
    Polyline (19,111) (19,129) (10,129) (24,150) (39,129) (29,129) (29,111), invisible if: NOT fbFunction.HW_Outputs.LiftDown
    Ellipse (65,82 17x17), colour toggle: fbFunction.CtrlOut.MagazineFull
    Label (84,83 77x16), "Magazine full"
    Ellipse (65,101 17x17), colour toggle: fbFunction.CtrlOut.PalletLifted
    Label (84,102 77x16), "Pallet Lifted"
    Ellipse (65,120 17x17), colour toggle: fbFunction.CtrlOut.StatusReady
    Label (84,121 77x16), "Status ready"
    Ellipse (65,139 17x17), colour toggle: fbFunction.CtrlOut.TransportEnabled
    Label (84,140 77x16), "Transport en."
END_VISUALIZATION

// ---- 20_Product/20_ProBox/40_TC_Visualization/11_Addon/ProfileCheckAddon/V_ProfileCheckAddon.TcVIS
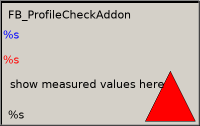
VISUALIZATION V_ProfileCheckAddon  // 200x126
VAR_IN_OUT
	{attribute 'VAR_IN_OUT_AS_POINTER'}
	fbFunction		: FB_ProfileCheckAddon;
END_VAR
    Rectangle (0,1 200x125)
    Rectangle (5,105 143x20), "%s", text variable: fbFunction.ConfigFunction.FunctionName
    Label (5,5 158x20), "FB_ProfileCheckAddon"
    Rectangle (0,25 99x20), "%s", text variable: fbFunction.ProfileCheckState.eState
    Polygon (145,121) (170,71) (195,121) (180,121) (160,121), invisible if: fbFunction.FunctionData.ErrorData.ErrorState = E_ErrorState.OPERATIONAL
    Rectangle (0,50 161x20), "%s", text variable: fbFunction.FunctionData.ErrorData.Error.ErrorCode.Conv, invisible if: fbFunction.FunctionData.ErrorData.Error.ErrorCode.Conv = 0
    Label (7,77 158x15), "show measured values here"
END_VISUALIZATION

// ---- 20_Product/20_ProBox/40_TC_Visualization/11_Addon/RejectPanelAddon/V_RejectPanelAddon.TcVIS
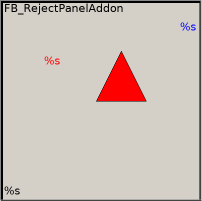
VISUALIZATION V_RejectPanelAddon  // 202x201
VAR_IN_OUT
	{attribute 'VAR_IN_OUT_AS_POINTER'}
	fbFunction		: FB_RejectPanelAddon;	
END_VAR
    Rectangle (1,1 200x200)
    Label (1,1 200x15), "FB_RejectPanelAddon"
    Rectangle (1,181 200x20), "%s", text variable: fbFunction.ConfigFunction.FunctionName
    Rectangle (41,51 161x20), "%s", text variable: fbFunction.ZoneData[1].ErrorData.Error.ErrorCode.Conv, invisible if: fbFunction.FunctionData.ErrorData.Error.ErrorCode.Conv = 0
    Polygon (96,101) (121,51) (146,101) (131,101) (111,101), invisible if: fbFunction.FunctionData.ErrorData.ErrorState = E_ErrorState.OPERATIONAL
    Rectangle (38,17 161x20), "%s", text variable: fbFunction.RejectPanelState.eState
END_VISUALIZATION

// ---- 20_Product/20_ProBox/40_TC_Visualization/11_Addon/SickScannerAddon/V_SickScannerAddon.TcVIS
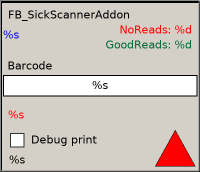
VISUALIZATION V_SickScannerAddon  // 200x172
VAR_IN_OUT
	{attribute 'VAR_IN_OUT_AS_POINTER'}
	fbFunction		: FB_SickScannerAddon;
END_VAR
    Rectangle (0,1 200x171)
    Rectangle (6,150 143x20), "%s", text variable: fbFunction.ConfigFunction.FunctionName
    Label (5,5 139x20), "FB_SickScannerAddon"
    Rectangle (0,25 99x20), "%s", text variable: fbFunction.BaseFunctionData.State.eState
    Rectangle (3,75 194x21), "%s", text variable: fbFunction.BaseFunctionData.LabelData.Label
    Polygon (155,166) (175,130) (195,166) (185,166) (165,166), invisible if: fbFunction.FunctionData.ErrorData.ErrorState = E_ErrorState.OPERATIONAL
    Rectangle (95,35 100x20), "GoodReads: %d", tooltip "good read counter", text variable: fbFunction.FunctionData.AddOnData.Counter[1]
    Rectangle (95,20 100x20), "NoReads: %d", tooltip "no read counter", text variable: fbFunction.FunctionData.AddOnData.Counter[2]
    Rectangle (5,105 192x20), "%s", tooltip "%s", text variable: fbFunction.FunctionData.ErrorData.Error.ErrorCode.Conv, invisible if: fbFunction.FunctionData.ErrorData.Error.ErrorCode.Conv = 0
        p4168582468: fbFunction.FunctionData.ErrorData.Error.ErrorParam
    Label (4,51 52x30), "Barcode"
    Checkbox (8,129 97x22), "Debug print", variable: fbFunction.BaseFunctionData.LabelData.DebugPrint
END_VISUALIZATION

// ---- 20_Product/20_ProBox/40_TC_Visualization/11_Addon/TLB4WeightAddon/V_TLB4WeightAddon.TcVIS
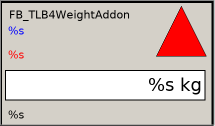
VISUALIZATION V_TLB4WeightAddon  // 215x126
VAR_IN_OUT
	{attribute 'VAR_IN_OUT_AS_POINTER'}
	fbFunction		: FB_TLB4WeightAddon;
END_VAR
    Rectangle (0,1 213x125)
    Rectangle (5,105 143x20), "%s", text variable: fbFunction.ConfigFunction.FunctionName
    Label (6,5 209x20), "FB_TLB4WeightAddon"
    Rectangle (5,21 99x20), "%s", text variable: fbFunction.WeightStates.eState
    Rectangle (5,70 200x30), "%s kg", text variable: fbFunction.Weight
    Polygon (156,56) (181,6) (206,56) (191,56) (171,56), invisible if: fbFunction.FunctionData.ErrorData.ErrorState = E_ErrorState.OPERATIONAL
    Rectangle (5,45 161x20), "%s", text variable: fbFunction.FunctionData.ErrorData.Error.ErrorCode.Conv, invisible if: fbFunction.FunctionData.ErrorData.Error.ErrorCode.Conv = 0
END_VISUALIZATION

// ---- 20_Product/20_ProBox/40_TC_Visualization/12_Functions/FunctionForks/V_FunctionFork.TcVIS
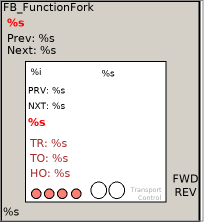
VISUALIZATION V_FunctionFork  // 204x222
VAR_INPUT
	ZoneIx : INT;
END_VAR

VAR_IN_OUT	
	{attribute 'VAR_IN_OUT_AS_POINTER'}
	fbFunction		: FB_FunctionForks;		
END_VAR
    Rectangle (0,0 200x222), colour toggle: fbFunction.BaseFunctionData.ZoneOrders[ZoneIx].Drive_Run OR fbFunction.BaseFunctionData.ZoneOrders[ZoneIx].Drive_RunRev
    Label (168,172 35x14), "FWD", invisible if: NOT fbFunction.BaseFunctionData.ZoneOrders[ZoneIx].Drive_Run
    Rectangle (0,204 200x16), "%s", text variable: fbFunction.ConfigFunction.Zone[ZoneIx].ZoneName
    Label (168,183 35x19), "REV", invisible if: NOT fbFunction.BaseFunctionData.ZoneOrders[ZoneIx].Drive_RunRev
    Label (0,0 200x15), "FB_FunctionFork"
    Rectangle (4,15 194x16), "%s", tooltip "%s", text variable: fbFunction.FunctionData.ErrorData.Error.ErrorCode.Conv, invisible if: fbFunction.FunctionData.ErrorData.ErrorState = E_ErrorState.OPERATIONAL
        p4168582468: fbFunction.FunctionData.ErrorData.Error.ErrorParam
    Frame (14,55 152x147)
        shows V_TransportControl(TransportControl := fbFunction.fbTransportControl, ZoneData := fbFunction.ZoneData[ZoneIx])
    Rectangle (4,32 200x13), "Prev: %s", tooltip "FunctionInterface.in.ePrevFunctionNumber", text variable: fbFunction.FunctionInterface.In.ePrevFunctionNumber
    Rectangle (4,44 200x13), "Next: %s", tooltip "FunctionInterface.in.eNextFunctionNumber", text variable: fbFunction.FunctionInterface.In.eNextFunctionNumber
END_VISUALIZATION

// ---- 20_Product/20_ProBox/40_TC_Visualization/12_Functions/LowLiftUnit/V_LowLiftUnit.TcVIS
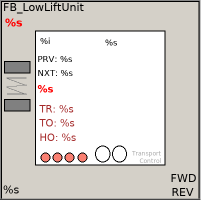
VISUALIZATION V_LowLiftUnit  // 201x200
VAR_IN_OUT
	{attribute 'VAR_IN_OUT_AS_POINTER'}
	fbFunction		: FB_LowLiftUnit;	
END_VAR
    Rectangle (0,0 200x200), colour toggle: fbFunction.BaseFunctionData.ZoneOrders[1].Drive_Run OR fbFunction.BaseFunctionData.ZoneOrders[1].Drive_RunRev
    Rectangle (0,180 200x20), "%s", text variable: fbFunction.ConfigFunction.FunctionName
    Label (0,0 200x15), "FB_LowLiftUnit"
    Label (166,172 35x13), "FWD", invisible if: NOT fbFunction.BaseFunctionData.ZoneOrders[1].Drive_Run
    Label (165,185 35x15), "REV", invisible if: NOT fbFunction.BaseFunctionData.ZoneOrders[1].Drive_RunRev
    Frame (25,25 140x140)
        shows V_TransportControl(TransportControl := fbFunction.fbTransportControl, ZoneData := fbFunction.ZoneData[1])
    Polyline (26,78) (7,78) (26,85) (7,87) (26,94) (7,94), colour toggle: fbFunction.HW_Outputs.Drive_Run_Up OR fbFunction.HW_Outputs.Drive_Run_Down
    Rectangle (4,99 26x12), tooltip "Lower lift sensor", colour toggle: fbFunction.HW_Inputs.Sensor_Pos_Down
    Rectangle (4,61 26x12), tooltip "Upper lift sensor", colour toggle: fbFunction.HW_Inputs.Sensor_Pos_Up
    Rectangle (2,15 194x16), "%s", tooltip "%s", text variable: fbFunction.FunctionData.ErrorData.Error.ErrorCode.Conv, invisible if: fbFunction.FunctionData.ErrorData.ErrorState = E_ErrorState.OPERATIONAL
        p4168582468: fbFunction.FunctionData.ErrorData.Error.ErrorParam
END_VISUALIZATION

// ---- 20_Product/20_ProBox/40_TC_Visualization/12_Functions/ProBoxStraightTransport/V_ProBoxStraightTransport.TcVIS
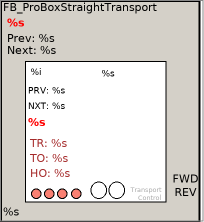
VISUALIZATION V_ProBoxStraightTransport  // 204x222
VAR_INPUT
	ZoneIx			: INT;
END_VAR

VAR_IN_OUT	
	{attribute 'VAR_IN_OUT_AS_POINTER'}
	fbFunction		: FB_ProBoxStraightTransport;		
END_VAR
    Rectangle (0,0 200x222), colour toggle: fbFunction.BaseFunctionData.ZoneOrders[ZoneIx].Drive_Run OR fbFunction.BaseFunctionData.ZoneOrders[ZoneIx].Drive_RunRev
    Label (168,172 35x14), "FWD", invisible if: NOT fbFunction.BaseFunctionData.ZoneOrders[ZoneIx].Drive_Run
    Rectangle (0,204 200x16), "%s", text variable: fbFunction.ConfigFunction.Zone[ZoneIx].ZoneName
    Label (168,183 35x19), "REV", invisible if: NOT fbFunction.BaseFunctionData.ZoneOrders[ZoneIx].Drive_RunRev
    Label (0,0 200x15), "FB_ProBoxStraightTransport"
    Rectangle (4,15 194x16), "%s", tooltip "%s", text variable: fbFunction.FunctionData.ErrorData.Error.ErrorCode.Conv, invisible if: fbFunction.FunctionData.ErrorData.ErrorState = E_ErrorState.OPERATIONAL
        p4168582468: fbFunction.FunctionData.ErrorData.Error.ErrorParam
    Frame (14,55 152x147)
        shows V_TransportControl(TransportControl := fbFunction.fbTransportControl[ZoneIx], ZoneData := fbFunction.ZoneData[ZoneIx])
    Rectangle (4,32 200x13), "Prev: %s", tooltip "FunctionInterface.in.ePrevFunctionNumber", text variable: fbFunction.FunctionInterface.In.ePrevFunctionNumber
    Rectangle (4,44 200x13), "Next: %s", tooltip "FunctionInterface.in.eNextFunctionNumber", text variable: fbFunction.FunctionInterface.In.eNextFunctionNumber
END_VISUALIZATION

// ---- 20_Product/20_ProBox/40_TC_Visualization/12_Functions/TransferCC/V_TransferCC.TcVIS
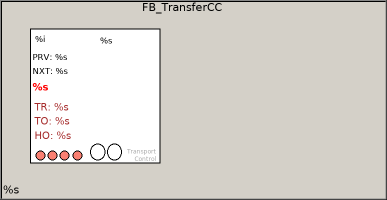
VISUALIZATION V_TransferCC  // 387x200
VAR_IN_OUT
	{attribute 'VAR_IN_OUT_AS_POINTER'}
	fbFunction		: FB_TransferCC;	
END_VAR
    Rectangle (0,0 387x200), colour toggle: fbFunction.BaseFunctionData.ZoneOrders[1].Drive_Run OR fbFunction.BaseFunctionData.ZoneOrders[1].Drive_RunRev
    Rectangle (0,180 200x20), "%s", text variable: fbFunction.ConfigFunction.FunctionName
    Label (139,0 107x15), "FB_TransferCC"
    Frame (20,23 140x140)
        shows V_TransportControl(TransportControl := fbFunction.fbTransportControl, ZoneData := fbFunction.ZoneData[1])
        p3560616238: SEL(fbFunction.HW_Inputs.Sensor_Pos_Left,SEL(fbFunction.HW_Inputs.Sensor_Pos_Right,100,0),200)
END_VISUALIZATION

// ---- 20_Product/20_ProBox/40_TC_Visualization/12_Functions/TransferUnit/V_TransferUnit.TcVIS
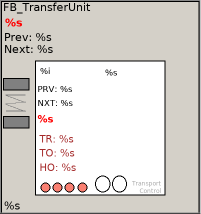
VISUALIZATION V_TransferUnit  // 201x214
VAR_IN_OUT
	{attribute 'VAR_IN_OUT_AS_POINTER'}
	fbFunction		: FB_TransferUnit;	
END_VAR
    Rectangle (0,0 200x214), colour toggle: fbFunction.Outputs.Drive_Run_12 OR fbFunction.Outputs.Drive_Run_21 OR fbFunction.Outputs.Drive_Run_34 OR fbFunction.Outputs.Drive_Run_43
    Rectangle (1,198 200x16), "%s", text variable: fbFunction.ConfigFunction.Zone[1].ZoneName
    Label (0,0 200x15), "FB_TransferUnit"
    Frame (25,55 140x140)
        shows V_TransportControl(TransportControl := fbFunction.fbTransportControl, ZoneData := fbFunction.ZoneData[1])
    Rectangle (2,15 196x16), "%s", tooltip "%s", text variable: fbFunction.FunctionData.ErrorData.Error.ErrorCode.Conv, invisible if: fbFunction.FunctionData.ErrorData.ErrorState = E_ErrorState.OPERATIONAL
        p4168582468: fbFunction.FunctionData.ErrorData.Error.ErrorParam
    Rectangle (3,116 26x12), tooltip "Lower lift sensor", colour toggle: fbFunction.HW_Inputs.Sensor_Pos_Down
    Rectangle (3,78 26x12), tooltip "Upper lift sensor", colour toggle: fbFunction.HW_Inputs.Sensor_Pos_Up
    Polyline (25,95) (6,95) (25,102) (6,104) (25,111) (6,111), colour toggle: fbFunction.HW_Outputs.Drive_Run_UpDown
    Rectangle (1,31 200x13), "Prev: %s", tooltip "FunctionInterface.in.ePrevFunctionNumber", text variable: fbFunction.FunctionInterface.In.ePrevFunctionNumber
    Rectangle (1,43 200x13), "Next: %s", tooltip "FunctionInterface.in.eNextFunctionNumber", text variable: fbFunction.FunctionInterface.In.eNextFunctionNumber
END_VISUALIZATION

// ---- 20_Product/20_ProBox/40_TC_Visualization/12_Functions/TurnTable/V_TurnTable.TcVIS
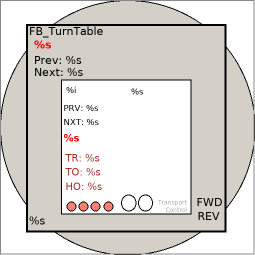
VISUALIZATION V_TurnTable  // 255x255
VAR_IN_OUT
	{attribute 'VAR_IN_OUT_AS_POINTER'}
	fbFunction		: FB_TurnTable;	
END_VAR
    Ellipse (0,0 255x255), colour toggle: fbFunction.FunctionInterface.Out.FunctionOrders.ReqDriveRun OR fbFunction.FunctionInterface.Out.FunctionOrders.ReqDriveRun_34
    Rectangle (26,24 200x208), colour toggle: fbFunction.HW_Outputs.Drive_Run_CW OR fbFunction.HW_Outputs.Drive_Run_CCW
    Rectangle (26,211 200x20), "%s", text variable: fbFunction.ConfigFunction.FunctionName
    Label (26,24 200x15), "FB_TurnTable"
    Label (192,196 35x13), "FWD", invisible if: NOT fbFunction.HW_Outputs.Drive_Run_CW
    Label (191,209 35x15), "REV", invisible if: NOT fbFunction.HW_Outputs.Drive_Run_CCW
    Frame (51,74 140x140)
        shows V_TransportControl(TransportControl := fbFunction.fbTransportControl, ZoneData := fbFunction.ZoneData[1])
    Rectangle (31,37 194x16), "%s", tooltip "%s", text variable: fbFunction.FunctionData.ErrorData.Error.ErrorCode.Conv, invisible if: fbFunction.FunctionData.ErrorData.ErrorState = E_ErrorState.OPERATIONAL
        p4168582468: fbFunction.FunctionData.ErrorData.Error.ErrorParam
    Rectangle (31,54 200x13), "Prev: %s", tooltip "FunctionInterface.in.ePrevFunctionNumber", text variable: fbFunction.FunctionInterface.In.ePrevFunctionNumber
    Rectangle (31,66 200x13), "Next: %s", tooltip "FunctionInterface.in.eNextFunctionNumber", text variable: fbFunction.FunctionInterface.In.eNextFunctionNumber
END_VISUALIZATION

// ---- 20_Product/20_ProBox/40_TC_Visualization/13_Elements/V_Element_Shuttle.TcVIS
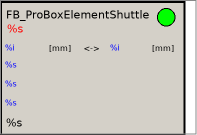
VISUALIZATION V_Element_Shuttle  // 197x135
VAR_IN_OUT
	{attribute 'VAR_IN_OUT_AS_POINTER'}
	fbFunction		: FB_ProBoxElementShuttle;
	//fbEmuFunction	: FB_ProBOXSG_Emulation;
END_VAR
    Rectangle (0,1 185x134), colour toggle: fbFunction.fbMpdControl.CtrlOut.MotionRunning
    Rectangle (3,113 143x20), "%s", text variable: fbFunction.ConfigElement.ElementName
    Label (3,5 158x20), "FB_ProBoxElementShuttle"
    Rectangle (2,38 54x20), "%i", tooltip "'Actual driver positon'", text variable: fbFunction.fbMpdControl._MPD.ActualPosValue
    Rectangle (4,19 161x20), "%s", tooltip "%s", text variable: fbFunction.ElementData.ErrorData.Error.ErrorCode.Conv, invisible if: fbFunction.ElementData.ErrorData.Error.ErrorCode.Conv = 0
        p4168582468: fbFunction.ElementData.ErrorData.Error.ErrorParam
    Rectangle (107,38 58x20), "%i", tooltip "'Set position'", text variable: fbFunction.fbMpdControl._MPD.RequestPosValue
        p4168582468: 'Set Position'
    Ellipse (157,8 18x18), colour toggle: NOT fbFunction.HW_Inputs.MotorUnitOK
    Label (45,42 30x13), "[mm]"
    Label (77,42 29x13), "<->"
    Rectangle (2,55 127x20), "%s", tooltip "'MPD State'", text variable: fbFunction.fbMpdControl._MPD.State
    Rectangle (2,74 195x20), "%s", text variable: fbFunction.fbMpdControl._MPD.CV[1].PickupFuncNumber
        p4168582468: 'PickupFuncNumber'
    Rectangle (2,93 183x20), "%s", text variable: fbFunction.fbMpdControl._MPD.CV[1].DepositFuncNumber
        p4168582468: 'DepositFuncNumber'
    Label (148,42 30x13), "[mm]"
END_VISUALIZATION

// ---- 20_Product/20_ProBox/40_TC_Visualization/13_Elements/V_Element_VC.TcVIS
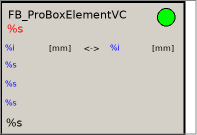
VISUALIZATION V_Element_VC  // 197x135
VAR_IN_OUT
	{attribute 'VAR_IN_OUT_AS_POINTER'}
	fbFunction		: FB_ProBoxElementVC;
	//fbEmuFunction	: FB_ProBOXSG_Emulation;
END_VAR
    Rectangle (0,1 185x134), colour toggle: fbFunction.fbMpdControl.CtrlOut.MotionRunning
    Rectangle (3,113 143x20), "%s", text variable: fbFunction.ConfigElement.ElementName
    Label (5,5 158x20), "FB_ProBoxElementVC"
    Rectangle (2,38 54x20), "%i", tooltip "'Actual driver positon'", text variable: fbFunction.fbMpdControl._MPD.ActualPosValue
    Rectangle (4,19 161x20), "%s", tooltip "%s", text variable: fbFunction.ElementData.ErrorData.Error.ErrorCode.Conv, invisible if: fbFunction.ElementData.ErrorData.Error.ErrorCode.Conv = 0
        p4168582468: fbFunction.ElementData.ErrorData.Error.ErrorParam
    Rectangle (107,38 58x20), "%i", tooltip "'Set position'", text variable: fbFunction.fbMpdControl._MPD.RequestPosValue
        p4168582468: 'Set Position'
    Ellipse (157,8 18x18), colour toggle: NOT fbFunction.HW_Inputs.MotorUnitOK
    Label (45,42 30x13), "[mm]"
    Label (77,42 29x13), "<->"
    Rectangle (2,55 127x20), "%s", tooltip "'MPD State'", text variable: fbFunction.fbMpdControl._MPD.State
    Rectangle (2,74 195x20), "%s", text variable: fbFunction.fbMpdControl._MPD.CV[1].PickupFuncNumber
        p4168582468: 'PickupFuncNumber'
    Rectangle (2,93 195x20), "%s", text variable: fbFunction.fbMpdControl._MPD.CV[1].DepositFuncNumber
        p4168582468: 'DepositFuncNumber'
    Label (148,42 30x13), "[mm]"
END_VISUALIZATION

